FUNCTION_BLOCK FB_CYLINDER_DA_TESTDEV2_4 IMPLEMENTS I_CYLINDER_DA_TESTDEV2_4
VAR_INPUT
  bDoableActing:                                          BOOL;
  lrCurrentPosAbs:                                        LREAL;
  rCurrentPressureInBar:                                  REAL;
  rCurrentPressureInBarA:                                 REAL;
  rCurrentPressureInBarB:                                 REAL;
  /// Cylinder piston surface A
  lrPistonSurfaceA:                                       LREAL;
  /// Cylinder piston surface B
  lrPistonSurfaceB:                                       LREAL;
  // Speed and Pressure regulation
  rSpeedRegulationFactor:                                 REAL;
  rSpeedRegulationTolerance:                              REAL;
  rPressureRegulationFactor:                              REAL;
  rPressureRegulationTolerance:                           REAL;
END_VAR
VAR //General
	{attribute 'instance-path'} 
  {attribute 'noinit'} 
	strInstancePath:									                      STRING;
	bInit: 												                          BOOL:=TRUE;
	strFullObjectPath: 								                      STRING;
	stEvent:											                          ST_EVENT;
	bAck:												                            BOOL;
END_VAR
VAR   // From FB_init	
	itfLogEvents: 										                      I_HANDLE_EVENTS;
  itfOpMode:											                        I_OP_MODE;
  itfOpModeVisu:											                    I_OP_MODE_PAUSE_VISU;
  itfValve_CylCtrl:                                       I_VALVE_X_3_PROP;
  itfValve_LockA:                                         I_VALVE_X_2;
  itfValve_LockB:                                         I_VALVE_X_2;
  itfValve_PressureLimit:                                 I_PRV_PROP;
  rEndPosTol:                                             REAL;
  /// Volume flow in l/min or dm³/min
  rPumpVolumeFlow:                                        REAL; // Volumenstrom
  /// Pump efficiency factor (0,5-1)
  rPumpEfficiencyFactor:                                  REAL; // Wirkungsgrad
END_VAR                                      				
VAR	// Step chain control                				
  eSeq, eLastSeq, eNextSeq:					                      E_SEQ_CYLINDER; 
                  				
  //eActiveSeqState, eLastActiveSeqState:                 E_SEQ_GENERAL;
	(*
  iInternalSeqStateCase, iLastInternalSeqStateCase:       INT:=0;       
	tonDelay, tonTimeOut, tonStepTime:						          TON;
	tDelay:													                        TIME := T#100MS;
	tTimeOut:												                        TIME := T#100MS;
	tTimeOutExt:											                      TIME := T#100MS;
	bDelayActive, bTimeOutActiveQuit, bTimeOutActiveNoQuit:	BOOL;//Timer Option
	bActiveStep, bDebugAcitve, bDebugNext:					        BOOL;//Debug Option
	i:														                          INT;
 	iError:													                        INT; //ERROR-CODE                    	                   		
	listLastSteps:											                    ARRAY[0..49] OF ST_LAST_STEPS;	
	strExtraInfo:											                      STRING; 
	eStep_Type:												                      E_STEP_STATE_TYPE; 
	bDebugModeActive:										                    BOOL;   
	bWaitForBreakpoint:										                  BOOL;
	bBreakpointActive:										                  BOOL;
	bDebugResume:											                      BOOL;   
	listBreakpoint:											                    ARRAY[0..10] OF  INT;    
*)
i:														                            INT;
ii:														                            INT;
iii:														                          INT;
stSeqCtrlGeneral:											                    ST_SEQ_CTRL_GEN;     	
END_VAR                                             		
VAR                                                 		
	bMethodeFromExtStarted:									                BOOL;
	bMethodeFromExtActive:									                BOOL;
	bMethodeFromExtDone:									                  BOOL;
	strTemp:												                        STRING;
END_VAR   
VAR
  stHMI:                                                  ST_HMI_CYLINDER;
  lrToSetPos:                                             LREAL;
  rTargetPressureInBarA:                                  REAL;
  rTargetPressureInBarB:                                  REAL;
  rTargetPressureInForceA:                                REAL;
  rTargetPressureInForceB:                                REAL;
  rTargetPressureInPercentA:                              REAL;
  rTargetPressureInPercentB:                              REAL;
  iTargetPressureAsValueA:                                INT;
  iTargetPressureAsValueB:                                INT;
  rSpeedInPercentToSet:                                   REAL;
  rSpeedInMmPerSToSet:                                    REAL;
  rCurrentSpeedInMmPerS:                                  REAL;
  bStrokeLengthInitialized:                               BOOL;
  rStrokeLength:                                          REAL;
  lrPos:                                                  LREAL;
  lrPosZero:                                              LREAL;
  lrPosMax:                                               LREAL;
  bOpenChA:                                               BOOL;
	bOpenChB:                                               BOOL;
END_VAR
VAR // Recording
  stRecord:											                          ST_RECORD;	 
	tonSaveInterval:											                  TON; 
	iCntRecord:											                        INT;	
	listGainRampData:									                      ARRAY[0..499] OF stMesswerte;
	stCurrentRamp:										                      stRampAnalytic;
	iCycleCntNormal:									                      INT;	
	uiLinRegStart:										                      UINT:=0;
  uiLinRegEnd:										                        UINT:=299; 
  rGainLimit_EndPos:                                      REAL:=0.1;
  lrLastPos:                                              LREAL;
  bJogCtrlBusy:                                           BOOL;
  bStartHPTrigger:                                        BOOL;
  bStartWPTrigger:                                        BOOL;
  bStopTrigger:                                           BOOL;
  bStartCalibrationClicked:                               BOOL;
  // Speed
  listPosTable:                                           ARRAY[1..100] OF REAL;
  lrTotalPath:                                            LREAL;
  x:                                                      INT;
  xx:                                                     INT;
  iCorrectedSpeedValue:                                   INT;
  rCorrectedSpeedPercent:                                 REAL;
  bRegulation:                                            BOOL;
  bRegulationTrigger:                                     BOOL;
  uiRegulationSeq:                                        UINT := 0;
  bCorrectionTrigger:                                     BOOL;
  bRegulationBusy:                                        BOOL;
  rCurrentForceInKN:                                      REAL;
  rCurrentForceInN:                                       REAL;
  rActiveForce:                                           REAL;
  iCorrectedPressureAsValue:                              INT;
  bPressureRegulationTrigger:                             BOOL;
  bPressureRegulationBusy:                                BOOL;
  bPressureCorrectionTrigger:                             BOOL;
  uiPressureRegulationSeq:                                UINT := 0;
  bPressureRegulation:                                    BOOL;
END_VAR                	
VAR_TEMP                    	
	iTemp:										                              INT;
END_VAR
VAR PERSISTENT
	listCylCalibration:                                     ARRAY[1..2, 1..100] OF LREAL;
  listCalibrationTable:                                   ARRAY[1..7] OF ST_CYL_CALIBRATION;
END_VAR

// Set FBs and Interfaces ready after switch internal step
IF stSeqCtrlGeneral.iInternalSeqStateCase <> stSeqCtrlGeneral.iLastInternalSeqStateCase AND NOT stSeqCtrlGeneral.bExitSetReadyState THEN
  IF TRUE
  AND itfValve_CylCtrl.M_SetReady()
  AND itfValve_LockA.M_SetReady()
  AND itfValve_LockB.M_SetReady()
  AND itfValve_PressureLimit.M_SetReady()
  THEN
    stSeqCtrlGeneral.bExitSetReadyState := TRUE;
  ELSE
    RETURN;
  END_IF
END_IF

stSeqCtrlGeneral.strObjectPath := strInstancePath;
stSeqCtrlGeneral.strObject := F_CreateObjectName(strInstancePath);

rCurrentForceInKN := P_CurrentForceInKN;
rCurrentForceInN := P_CurrentForceInKN * 1000;

// First method call
_m_SequenceManager();
//_m_SaveLastStep();
_m_Recording();
_m_SpeedRegulation();
_m_PressureRegulation();
_m_PressureCalibration();
_m_HMI();

CASE eSeq OF 
  E_SEQ_CYLINDER.BASE:;
  
	E_SEQ_CYLINDER.INIT: _m_Seq_INIT();
		IF TRUE
		AND (stSeqCtrlGeneral.eActiveSeqState = E_SEQ_GENERAL.DONE) 
		THEN
			eSeq := E_SEQ_CYLINDER.BASE;
		END_IF
		
	E_SEQ_CYLINDER.SETUP:;
  
	// Process
  E_SEQ_CYLINDER.SET_MAX_POS: _m_Seq_SET_MAX_POS();
    IF TRUE
		AND (stSeqCtrlGeneral.eActiveSeqState = E_SEQ_GENERAL.DONE) 
		THEN
			eSeq := E_SEQ_CYLINDER.BASE;
		END_IF
  
  E_SEQ_CYLINDER.SET_WORK_PRESSURE: _m_Seq_SET_WORK_PRESSURE();
    IF TRUE
		AND (stSeqCtrlGeneral.eActiveSeqState = E_SEQ_GENERAL.DONE) 
		THEN
			eSeq := E_SEQ_CYLINDER.BASE;
		END_IF
  
  E_SEQ_CYLINDER.SET_ZERO_POS: _m_Seq_SET_ZERO_POS();
    IF TRUE
		AND (stSeqCtrlGeneral.eActiveSeqState = E_SEQ_GENERAL.DONE) 
		THEN
			eSeq := E_SEQ_CYLINDER.BASE;
		END_IF
  
  E_SEQ_CYLINDER.STOP: _m_Seq_STOP();
    IF TRUE
		AND (stSeqCtrlGeneral.eActiveSeqState = E_SEQ_GENERAL.DONE) 
		THEN
			eSeq := E_SEQ_CYLINDER.BASE;
		END_IF
    
  E_SEQ_CYLINDER.STOP_AND_LOCK: _m_Seq_STOP_AND_LOCK();
    IF TRUE
		AND (stSeqCtrlGeneral.eActiveSeqState = E_SEQ_GENERAL.DONE) 
		THEN
			eSeq := E_SEQ_CYLINDER.BASE;
		END_IF
  
  E_SEQ_CYLINDER.TO_HP: _m_Seq_TO_HP();
    IF TRUE
		AND (stSeqCtrlGeneral.eActiveSeqState = E_SEQ_GENERAL.DONE) 
		THEN
			eSeq := E_SEQ_CYLINDER.BASE;
		END_IF
  
  E_SEQ_CYLINDER.TO_SET_POS: _m_Seq_TO_SET_POS();
    IF TRUE
		AND (stSeqCtrlGeneral.eActiveSeqState = E_SEQ_GENERAL.DONE) 
		THEN
			eSeq := E_SEQ_CYLINDER.BASE;
		END_IF
  
  E_SEQ_CYLINDER.TO_WP: _m_Seq_TO_WP();
    IF TRUE
		AND (stSeqCtrlGeneral.eActiveSeqState = E_SEQ_GENERAL.DONE) 
		THEN
			eSeq := E_SEQ_CYLINDER.BASE;
		END_IF
    
  E_SEQ_CYLINDER.PRESSURE_CALIBRATION: _m_Seq_PRESSURE_CALIBRATION();
    IF TRUE
		AND (stSeqCtrlGeneral.eActiveSeqState = E_SEQ_GENERAL.DONE) 
		THEN
			eSeq := E_SEQ_CYLINDER.BASE;
		END_IF
    
  E_SEQ_CYLINDER.OPEN_LOCK_VALVES: _m_Seq_OPEN_LOCK_VALVES();
    IF TRUE
		AND (stSeqCtrlGeneral.eActiveSeqState = E_SEQ_GENERAL.DONE) 
		THEN
			eSeq := E_SEQ_CYLINDER.BASE;
		END_IF

  // End
	E_SEQ_CYLINDER.END:;
	E_SEQ_CYLINDER.ERROR_SEQ:;	
END_CASE

strTemp:=TO_STRING(eSeq);

METHOD PRIVATE _m_DebugManager
VAR_INPUT
	iStepID: int;
END_VAR
IF TRUE
AND THIS^.stSeqCtrlGeneral.bDebugModeActive 
AND NOT THIS^.stSeqCtrlGeneral.bActiveStep
THEN


THIS^.stSeqCtrlGeneral.bBreakpointActive:=FALSE;

FOR i:=0 TO 10 DO
	
	IF TRUE
	AND iStepID=THIS^.stSeqCtrlGeneral.listBreakpoint[i] 
	AND iStepID<>0
	THEN
		EXIT;
	END_IF
END_FOR
IF (i<=10) THEN
	THIS^.stSeqCtrlGeneral.bBreakpointActive:=TRUE;
END_IF

END_IF
END_METHOD

METHOD PRIVATE _m_Delay : BOOL
VAR_INPUT
	DelayTime:	TIME;
END_VAR
THIS^.stSeqCtrlGeneral.bDelayActive:=TRUE;
THIS^.stSeqCtrlGeneral.tDelay:=DelayTime;
_m_Delay:=FALSE;
IF THIS^.stSeqCtrlGeneral.tonDelay.Q THEN
	_m_Delay:=TRUE;
END_IF
END_METHOD

METHOD PRIVATE _m_GeneralStepSetting : BOOL
VAR_INPUT
	StepType:			    	E_STEP_STATE_TYPE;
	InfoTextID:					STRING(20);
	EnableDebug:	   			BOOL;	
	
END_VAR
IF THIS^.stSeqCtrlGeneral.bActiveStep THEN
	THIS^.stSeqCtrlGeneral.eStep_Type:=StepType;
	THIS^.stSeqCtrlGeneral.strExtraInfo:= GenLib.F_RET_TXTLIST_ENTRY(strPortNr:='851',strID:='',strTxtLstName:=InfoTextID);
END_IF
END_METHOD

METHOD PRIVATE _m_HMI : BOOL
VAR_INPUT
END_VAR
THIS^.stHMI.bInHP := THIS^.lrPos <= 1;
THIS^.stHMI.bInWP := THIS^.lrPos >= rStrokeLength - 1;
THIS^.stHMI.bPressureOk := THIS^.rCurrentPressureInBar > 25;
THIS^.stHMI.lrCurrentPos := THIS^.lrPos;
THIS^.stHMI.lrMaxPosVal := THIS^.lrPosMax;
THIS^.stHMI.lrMinPosVal := THIS^.lrPosZero;
THIS^.stHMI.sState := TO_STRING(THIS^.eSeq);
END_METHOD

METHOD PRIVATE _m_ManualOperation : BOOL
VAR_INPUT
END_VAR
IF TRUE 
AND THIS^.itfOpMode.P_OP_MODE_STATE = OP_MODE.MANUAL 
AND THIS^.itfOpModeVisu.P_HandSelected
AND THIS^.stHMI.bToHPTriggered
AND NOT THIS^.bJogCtrlBusy
THEN
  THIS^.stSeqCtrlGeneral.eActiveSeqState := E_SEQ_GENERAL.READY;
  THIS^.bStartHPTrigger := TRUE;
  THIS^.bJogCtrlBusy := TRUE;
ELSIF TRUE 
AND THIS^.itfOpMode.P_OP_MODE_STATE = OP_MODE.MANUAL 
AND THIS^.itfOpModeVisu.P_HandSelected
AND THIS^.stHMI.bToWPTriggered
AND NOT THIS^.bJogCtrlBusy
THEN
  THIS^.stSeqCtrlGeneral.eActiveSeqState := E_SEQ_GENERAL.READY;
  THIS^.bStartWPTrigger := TRUE;
  THIS^.bJogCtrlBusy := TRUE; 
ELSIF TRUE 
AND THIS^.itfOpMode.P_OP_MODE_STATE = OP_MODE.MANUAL 
AND THIS^.itfOpModeVisu.P_HandSelected
AND THIS^.stHMI.bToSetPosTriggered
AND NOT THIS^.bJogCtrlBusy
THEN
  //M_ToSetPos(lrToSetPos:= 500, rSpeedInPercent:= 100);
  THIS^.bJogCtrlBusy := TRUE;
ELSIF TRUE 
AND THIS^.itfOpMode.P_OP_MODE_STATE = OP_MODE.MANUAL 
AND THIS^.itfOpModeVisu.P_HandSelected
AND NOT THIS^.stHMI.bToHPTriggered
AND NOT THIS^.stHMI.bToWPTriggered
AND NOT THIS^.stHMI.bToSetPosTriggered
AND THIS^.bJogCtrlBusy
THEN
  THIS^.stSeqCtrlGeneral.eActiveSeqState := E_SEQ_GENERAL.READY;
  THIS^.bStopTrigger := TRUE;
  THIS^.bStartHPTrigger := FALSE;
  THIS^.bStartWPTrigger := FALSE;
  THIS^.bJogCtrlBusy := FALSE;
END_IF



IF THIS^.bStartWPTrigger THEN
  IF M_ToWP(ePressureType:= E_PRESSURE_TYPE.PERCENT, rWorkPressure:= 50, eSpeedType:= E_SPEED_TYPE.PERCENT, rSpeed:= 100) THEN
    THIS^.bStartWPTrigger := FALSE;
	END_IF
END_IF
IF THIS^.bStartHPTrigger THEN
  IF M_ToHP(ePressureType:= E_PRESSURE_TYPE.PERCENT, rWorkPressure:= 50, eSpeedType:= E_SPEED_TYPE.PERCENT, rSpeed:= 100) THEN
    THIS^.bStartHPTrigger := FALSE;
	END_IF
END_IF
IF THIS^.bStopTrigger THEN
  IF M_Stop() THEN
    THIS^.bStopTrigger := FALSE;
	END_IF
END_IF
END_METHOD

METHOD PRIVATE _m_PressureCalibration : BOOL
VAR_INPUT
END_VAR
// Calibration clicked
IF TRUE
AND THIS^.itfOpMode.P_OP_MODE_STATE = OP_MODE.MANUAL 
AND THIS^.bStartCalibrationClicked 
THEN
  IF M_PressureCalibration() THEN
    THIS^.stSeqCtrlGeneral.eActiveSeqState := E_SEQ_GENERAL.READY;
    THIS^.bStartCalibrationClicked := FALSE;
	END_IF
END_IF
END_METHOD

(******************Description****************)
// This function allows variable pressure control
(*********************************************)
METHOD PRIVATE _m_PressureRegulation : BOOL
VAR_INPUT
END_VAR
IF TRUE
AND THIS^.rCurrentForceInN < THIS^.rActiveForce 
AND THIS^.iCorrectedPressureAsValue < 32768
AND THIS^.bPressureRegulationTrigger
AND NOT THIS^.bPressureRegulationBusy
THEN
  IF ABS(THIS^.rCurrentForceInN - THIS^.rActiveForce) > THIS^.rPressureRegulationTolerance THEN
    //THIS^.iCorrectedPressureAsValue := THIS^.iCorrectedPressureAsValue + 100;
    THIS^.iCorrectedPressureAsValue := TO_INT(THIS^.iCorrectedPressureAsValue + ABS((THIS^.rCurrentForceInN - THIS^.rActiveForce) * THIS^.rPressureRegulationFactor));
    THIS^.bPressureCorrectionTrigger := TRUE;
  END_IF
ELSIF TRUE
AND THIS^.rCurrentForceInN > THIS^.rActiveForce 
AND THIS^.iCorrectedPressureAsValue > 0
AND THIS^.bPressureRegulationTrigger
AND NOT THIS^.bPressureRegulationBusy
THEN
  IF ABS(THIS^.rCurrentForceInN - THIS^.rActiveForce) > THIS^.rPressureRegulationTolerance THEN
    //THIS^.iCorrectedPressureAsValue := THIS^.iCorrectedPressureAsValue - 100;
    THIS^.iCorrectedPressureAsValue := TO_INT(THIS^.iCorrectedPressureAsValue - ABS((THIS^.rCurrentForceInN - THIS^.rActiveForce) * THIS^.rPressureRegulationFactor));
    THIS^.bPressureCorrectionTrigger := TRUE;
  END_IF
END_IF

// Set Valve value correction
IF THIS^.bPressureCorrectionTrigger THEN
  THIS^.bPressureRegulationBusy:= TRUE;
  CASE THIS^.uiPressureRegulationSeq OF
    0:;
      IF THIS^.itfValve_PressureLimit.M_SetReady() THEN
        THIS^.uiPressureRegulationSeq := 1;
	    END_IF
    1:;
      IF THIS^.itfValve_PressureLimit.M_SetLimit(ePressureType:= E_PRESSURE_TYPE.VALUE, rLimit:= iCorrectedPressureAsValue) THEN
        THIS^.bPressureCorrectionTrigger := FALSE;
        THIS^.bPressureRegulationBusy := FALSE;
        THIS^.uiPressureRegulationSeq := 0;
	    END_IF
	END_CASE
END_IF
END_METHOD

METHOD PRIVATE _m_Recording : BOOL
VAR_INPUT
END_VAR
VAR
	i:                      DINT;
END_VAR
// Recording data for 5s
tonSaveInterval(IN:= NOT tonSaveInterval.Q, pt:= T#100MS);

IF iCntRecord > 499 OR iCntRecord < 0 THEN
	iCntRecord := 0;
END_IF

IF THIS^.tonSaveInterval.Q THEN
	FOR i := 299 TO 1 BY -1 DO
		THIS^.stRecord.listRecordData[i].rPosition := THIS^.stRecord.listRecordData[i - 1].rPosition;	                                  		
		THIS^.stRecord.listRecordData[i].rPressureInBar := THIS^.stRecord.listRecordData[i - 1].rPressureInBar;
	END_FOR		

	// Messergebnisse in Array eintragen	
	THIS^.stRecord.listRecordData[i].rPosition :=	THIS^.lrPos;
	THIS^.stRecord.listRecordData[i].rPressureInBar := THIS^.rCurrentPressureInBar;
END_IF

// Calibration table
FOR THIS^.iii := 1 TO 7 BY 1 DO
  THIS^.listCylCalibration[2, THIS^.iii] := TO_LREAL(THIS^.listCalibrationTable[THIS^.iii].uiValue);
  THIS^.listCylCalibration[1, THIS^.iii] := TO_LREAL(THIS^.listCalibrationTable[THIS^.iii].uiPressure);
END_FOR

// Position
THIS^.lrPos := -(THIS^.lrCurrentPosAbs / 1000 - THIS^.lrPosZero);
THIS^.rStrokeLength := -(THIS^.lrPosMax - THIS^.lrPosZero);

// Speed
IF THIS^.x < 1 OR THIS^.x > 100 THEN
  THIS^.x := 1;
END_IF
THIS^.listPosTable[THIS^.x] := THIS^.lrPos - THIS^.lrLastPos;
THIS^.lrTotalPath := 0;
FOR THIS^.xx := 1 TO 100 BY 1 DO
  THIS^.lrTotalPath := THIS^.lrTotalPath + THIS^.listPosTable[THIS^.xx];
END_FOR
THIS^.rCurrentSpeedInMmPerS := THIS^.lrTotalPath;
THIS^.x := THIS^.x + 1;
THIS^.lrLastPos := THIS^.lrPos;
END_METHOD

METHOD PRIVATE _m_SaveLastStep : BOOL
VAR_INPUT
END_VAR
VAR
	i: dint;
END_VAR
IF NOT THIS^.stSeqCtrlGeneral.bActiveStep THEN
	
	FOR i:=49 TO 1 BY -1 DO
			stSeqCtrlGeneral.listLastSteps[i].strStepName:=stSeqCtrlGeneral.listLastSteps[i-1].strStepName;
			stSeqCtrlGeneral.listLastSteps[i].tStepTime:=stSeqCtrlGeneral.listLastSteps[i-1].tStepTime;
			stSeqCtrlGeneral.listLastSteps[i].tDelayTime:=stSeqCtrlGeneral.listLastSteps[i-1].tDelayTime;
	END_FOR
	stSeqCtrlGeneral.listLastSteps[0].strStepName:=TO_STRING(THIS^.eSeq);
	stSeqCtrlGeneral.listLastSteps[1].tStepTime:=THIS^.stSeqCtrlGeneral.tonStepTime.ET;
	stSeqCtrlGeneral.listLastSteps[1].tStepTime:=THIS^.stSeqCtrlGeneral.tonDelay.ET;
ELSE
	stSeqCtrlGeneral.listLastSteps[0].tStepTime:=THIS^.stSeqCtrlGeneral.tonStepTime.ET;
	stSeqCtrlGeneral.listLastSteps[0].tDelayTime:=THIS^.stSeqCtrlGeneral.tonDelay.ET;	
END_IF
END_METHOD

METHOD PRIVATE _m_Seq_INIT : E_SEQ_PROCESS
VAR_INPUT
END_VAR
VAR
	ActiveSeq: STRING;
END_VAR
VAR
	i:         INT;
END_VAR
//THIS^._m_GeneralStepSetting(StepType:=E_STEP_STATE_TYPE.INIT,
ActiveSeq := TO_STRING(THIS^.eSeq);

CASE THIS^.stSeqCtrlGeneral.eActiveSeqState OF
E_SEQ_GENERAL.READY:;

	
E_SEQ_GENERAL.EXECUTE:;
	IF TRUE
	THEN
		THIS^.stSeqCtrlGeneral.eActiveSeqState := E_SEQ_GENERAL.RESET;
	END_IF
E_SEQ_GENERAL.RESET:;
	stSeqCtrlGeneral.iInternalSeqStateCase := 0;
	IF TRUE
	THEN
		THIS^.stSeqCtrlGeneral.eActiveSeqState := E_SEQ_GENERAL.BUSY;
	END_IF
  
E_SEQ_GENERAL.BUSY:;
	CASE THIS^.stSeqCtrlGeneral.iInternalSeqStateCase OF
		0:	// Reset valves
      IF TRUE
      AND THIS^.itfValve_CylCtrl.M_Reset()
      AND THIS^.itfValve_LockA.M_ToHP(tDelay:= T#10MS)
      AND THIS^.itfValve_LockB.M_ToHP(tDelay:= T#10MS)
			THEN 
				THIS^.stSeqCtrlGeneral.iInternalSeqStateCase := 1000;
			END_IF
      
    1000: // Exit step
      IF TRUE
			THEN 
				THIS^.stSeqCtrlGeneral.iInternalSeqStateCase := 9999;
			END_IF
      
	ELSE
		THIS^.stSeqCtrlGeneral.eActiveSeqState := E_SEQ_GENERAL.DONE;  
	END_CASE
	THIS^.stSeqCtrlGeneral.strExtraInfo := CONCAT('Internal state: ', TO_STRING(THIS^.stSeqCtrlGeneral.iInternalSeqStateCase));
E_SEQ_GENERAL.DONE:;
E_SEQ_GENERAL.ERROR:;
E_SEQ_GENERAL.TIME_OUT:; 

IF TRUE
AND THIS^.stSeqCtrlGeneral.bTimeOutActiveQuit 
THEN
  THIS^.stSeqCtrlGeneral.strExtraInfo := 'Bitte quittieren und erneut testen';
  IF TRUE
  //AND itfOpMode.P_QUIT
  THEN
    THIS^.stSeqCtrlGeneral.eActiveSeqState := E_SEQ_GENERAL.EXECUTE;
	END_IF
  
END_IF

ELSE
  THIS^.stSeqCtrlGeneral.eActiveSeqState := E_SEQ_GENERAL.ERROR;
END_CASE
END_METHOD

METHOD PRIVATE _m_Seq_OPEN_LOCK_VALVES : E_SEQ_PROCESS
VAR_INPUT
END_VAR
VAR
	ActiveSeq: STRING;
END_VAR
VAR
	
END_VAR
//THIS^._m_GeneralStepSetting(StepType:=E_STEP_STATE_TYPE.INIT,
ActiveSeq := TO_STRING(THIS^.eSeq);

CASE THIS^.stSeqCtrlGeneral.eActiveSeqState OF
E_SEQ_GENERAL.READY:;

	
E_SEQ_GENERAL.EXECUTE:;
	IF TRUE
	THEN
		THIS^.stSeqCtrlGeneral.eActiveSeqState := E_SEQ_GENERAL.RESET;
	END_IF
  
E_SEQ_GENERAL.RESET:;
	stSeqCtrlGeneral.iInternalSeqStateCase := 0;
	IF TRUE
	THEN
		THIS^.stSeqCtrlGeneral.eActiveSeqState := E_SEQ_GENERAL.BUSY;
	END_IF
  
E_SEQ_GENERAL.BUSY:;
	CASE THIS^.stSeqCtrlGeneral.iInternalSeqStateCase OF
    0:	// Check if open A
      IF TRUE
			THEN 
        IF THIS^.bOpenChA THEN
          THIS^.stSeqCtrlGeneral.iInternalSeqStateCase := 10;
        ELSE
          THIS^.stSeqCtrlGeneral.iInternalSeqStateCase := 20;
        END_IF
			END_IF

    10:	// Open A
      IF TRUE 
      AND THIS^.itfValve_LockA.M_ToWP1(tDelay:= T#0MS)
			THEN 
        THIS^.stSeqCtrlGeneral.iInternalSeqStateCase := 30;
			END_IF
      
		20:	// Close A
      IF TRUE
      AND THIS^.itfValve_LockA.M_ToHP(tDelay:= T#0MS)
			THEN 
        THIS^.stSeqCtrlGeneral.iInternalSeqStateCase := 30;
			END_IF
      
    30:	// Check if open B
      IF TRUE
			THEN 
        IF THIS^.bOpenChB THEN
          THIS^.stSeqCtrlGeneral.iInternalSeqStateCase := 40;
        ELSE
          THIS^.stSeqCtrlGeneral.iInternalSeqStateCase := 50;
        END_IF
			END_IF

    40:	// Open B
      IF TRUE
      AND THIS^.itfValve_LockB.M_ToWP1(tDelay:= T#0MS)
			THEN 
        THIS^.stSeqCtrlGeneral.iInternalSeqStateCase := 1000;
			END_IF
      
		50:	// Close B
      IF TRUE
      AND THIS^.itfValve_LockB.M_ToHP(tDelay:= T#0MS)
			THEN 
        THIS^.stSeqCtrlGeneral.iInternalSeqStateCase := 1000;
			END_IF
      
    1000: // Exit step
      IF TRUE
			THEN 
				THIS^.stSeqCtrlGeneral.iInternalSeqStateCase := 9999;
			END_IF
      
	ELSE
		THIS^.stSeqCtrlGeneral.eActiveSeqState := E_SEQ_GENERAL.DONE;  
	END_CASE
	THIS^.stSeqCtrlGeneral.strExtraInfo := CONCAT('Internal state: ', TO_STRING(THIS^.stSeqCtrlGeneral.iInternalSeqStateCase));

E_SEQ_GENERAL.DONE:;

E_SEQ_GENERAL.ERROR:;

E_SEQ_GENERAL.TIME_OUT:; 
IF TRUE
AND THIS^.stSeqCtrlGeneral.bTimeOutActiveQuit 
THEN
  THIS^.stSeqCtrlGeneral.strExtraInfo := 'Bitte quittieren und erneut testen';
  IF TRUE
  //AND itfOpMode.P_QUIT
  THEN
    THIS^.stSeqCtrlGeneral.eActiveSeqState := E_SEQ_GENERAL.EXECUTE;
	END_IF
  
END_IF

ELSE
  THIS^.stSeqCtrlGeneral.eActiveSeqState := E_SEQ_GENERAL.ERROR;
END_CASE
END_METHOD

METHOD PRIVATE _m_Seq_PRESSURE_CALIBRATION : E_SEQ_PROCESS
VAR_INPUT
END_VAR
VAR
	ActiveSeq:  STRING;
END_VAR
//THIS^._m_GeneralStepSetting(StepType:=E_STEP_STATE_TYPE.INIT,
ActiveSeq := TO_STRING(THIS^.eSeq);

CASE THIS^.stSeqCtrlGeneral.eActiveSeqState OF
E_SEQ_GENERAL.READY:;

	
E_SEQ_GENERAL.EXECUTE:;
	IF TRUE
	THEN
		THIS^.stSeqCtrlGeneral.eActiveSeqState := E_SEQ_GENERAL.RESET;
	END_IF
  
E_SEQ_GENERAL.RESET:;
	stSeqCtrlGeneral.iInternalSeqStateCase := 0;
	IF TRUE
	THEN
    THIS^.ii := 1;
    FOR THIS^.ii := 1 TO 7 BY 1 DO
      THIS^.listCalibrationTable[THIS^.ii].uiValue := 0;
      THIS^.listCalibrationTable[THIS^.ii].uiPressure := 0;
      THIS^.listCalibrationTable[THIS^.ii].uiState := 0;
		END_FOR
    THIS^.ii := 1;
		THIS^.stSeqCtrlGeneral.eActiveSeqState := E_SEQ_GENERAL.BUSY;
	END_IF
  
E_SEQ_GENERAL.BUSY:;
	CASE THIS^.stSeqCtrlGeneral.iInternalSeqStateCase OF
		0:	// Set work pressure value to XXXX
      IF TRUE
      AND THIS^.itfValve_PressureLimit.M_SetLimit(ePressureType:= E_PRESSURE_TYPE.VALUE, rLimit:= 1000 * THIS^.ii)
			THEN 
        THIS^.listCalibrationTable[THIS^.ii].uiValue := TO_UINT(1000 * THIS^.ii);
        THIS^.listCalibrationTable[THIS^.ii].uiState := 1;
        THIS^.stSeqCtrlGeneral.iInternalSeqStateCase := 10;
			END_IF
      
    10:	// Open A channel
      IF TRUE
      AND THIS^.itfValve_LockA.M_ToWP1(tDelay:= T#10MS)
			THEN 
        IF THIS^.bDoableActing THEN
				  THIS^.stSeqCtrlGeneral.iInternalSeqStateCase := 20;
        ELSE
          THIS^.stSeqCtrlGeneral.iInternalSeqStateCase := 30;
        END_IF
			END_IF
      
    20:	// Open B channel
      IF TRUE
      AND THIS^.itfValve_LockB.M_ToWP1(tDelay:= T#10MS)
			THEN 
				THIS^.stSeqCtrlGeneral.iInternalSeqStateCase := 30;
			END_IF
      
    30: // Move cylinder to WP
      IF TRUE
      AND THIS^.itfValve_CylCtrl.M_ValveCtrl(rSpeedInPercent:= 100, tDelay:= T#10MS)
			THEN 
        THIS^.stSeqCtrlGeneral.iInternalSeqStateCase := 40;
			END_IF
      
    40: // Choice step
      IF TRUE
      THEN
        IF THIS^.ii = 1 THEN
          THIS^.stSeqCtrlGeneral.iInternalSeqStateCase := 50;
        ELSE
          THIS^.stSeqCtrlGeneral.iInternalSeqStateCase := 60;
				END_IF
			END_IF
      
    50: // Delay step (wait for cylinder end position)
      IF TRUE
      AND _m_Delay(DelayTime:= T#30S)
      THEN
        THIS^.stSeqCtrlGeneral.iInternalSeqStateCase := 60;
			END_IF
      
    60: // Delay step (cylinder under load)
      IF TRUE
      AND _m_Delay(DelayTime:= T#5S)
      THEN
        THIS^.stSeqCtrlGeneral.iInternalSeqStateCase := 70;
			END_IF
      
    70: // Save pressure
      IF TRUE
      THEN
        THIS^.listCalibrationTable[THIS^.ii].uiPressure := TO_UINT(THIS^.rCurrentPressureInBar);
        THIS^.listCalibrationTable[THIS^.ii].uiState := 2;
        THIS^.stSeqCtrlGeneral.iInternalSeqStateCase := 80;
			END_IF
      
    80: // Decide step
      IF TRUE
      AND _m_Delay(DelayTime:= T#1S)
      THEN
        IF THIS^.ii >= 7 OR THIS^.ii < 1 THEN
          THIS^.ii := 1;
          THIS^.stSeqCtrlGeneral.iInternalSeqStateCase := 1000;
        ELSE
          THIS^.ii := THIS^.ii + 1;
          THIS^.stSeqCtrlGeneral.iInternalSeqStateCase := 0;
				END_IF
			END_IF
      
    1000: // Stop and exit
      IF TRUE
      AND THIS^.itfValve_PressureLimit.M_SetLimit(ePressureType:= E_PRESSURE_TYPE.VALUE, rLimit:= 0)
      AND THIS^.itfValve_CylCtrl.M_ValveCtrl(rSpeedInPercent:= 0, tDelay:= T#10MS)
      AND THIS^.itfValve_LockA.M_ToHP(tDelay:= T#10MS)
      AND THIS^.itfValve_LockB.M_ToHP(tDelay:= T#10MS)
			THEN 
				THIS^.stSeqCtrlGeneral.iInternalSeqStateCase := 9999;
			END_IF
      
	ELSE
		THIS^.stSeqCtrlGeneral.eActiveSeqState := E_SEQ_GENERAL.DONE;  
	END_CASE
	THIS^.stSeqCtrlGeneral.strExtraInfo := CONCAT('Internal state: ', TO_STRING(THIS^.stSeqCtrlGeneral.iInternalSeqStateCase));

E_SEQ_GENERAL.DONE:;

E_SEQ_GENERAL.ERROR:;

E_SEQ_GENERAL.TIME_OUT:; 
IF TRUE
AND THIS^.stSeqCtrlGeneral.bTimeOutActiveQuit 
THEN
  THIS^.stSeqCtrlGeneral.strExtraInfo := 'Bitte quittieren und erneut testen';
  IF TRUE
  //AND itfOpMode.P_QUIT
  THEN
    THIS^.stSeqCtrlGeneral.eActiveSeqState := E_SEQ_GENERAL.EXECUTE;
	END_IF
  
END_IF

ELSE
  THIS^.stSeqCtrlGeneral.eActiveSeqState := E_SEQ_GENERAL.ERROR;
END_CASE
END_METHOD

METHOD PRIVATE _m_Seq_SET_MAX_POS : E_SEQ_PROCESS
VAR_INPUT
END_VAR
VAR
	ActiveSeq: STRING;
END_VAR
VAR
	
END_VAR
//THIS^._m_GeneralStepSetting(StepType:=E_STEP_STATE_TYPE.INIT,
ActiveSeq := TO_STRING(THIS^.eSeq);

CASE THIS^.stSeqCtrlGeneral.eActiveSeqState OF
E_SEQ_GENERAL.READY:;

	
E_SEQ_GENERAL.EXECUTE:;
	IF TRUE
	THEN
		THIS^.stSeqCtrlGeneral.eActiveSeqState := E_SEQ_GENERAL.RESET;
	END_IF
  
E_SEQ_GENERAL.RESET:;
	stSeqCtrlGeneral.iInternalSeqStateCase := 0;
	IF TRUE
	THEN
		THIS^.stSeqCtrlGeneral.eActiveSeqState := E_SEQ_GENERAL.BUSY;
	END_IF
  
E_SEQ_GENERAL.BUSY:;
	CASE THIS^.stSeqCtrlGeneral.iInternalSeqStateCase OF
		0:	// Set max position
      IF TRUE 
			THEN 
        THIS^.lrPosMax := THIS^.lrCurrentPosAbs / 1000;
        THIS^.stSeqCtrlGeneral.iInternalSeqStateCase := 1000;
			END_IF
      
    1000: // Exit step
      IF TRUE
			THEN 
				THIS^.stSeqCtrlGeneral.iInternalSeqStateCase := 9999;
			END_IF
      
	ELSE
		THIS^.stSeqCtrlGeneral.eActiveSeqState := E_SEQ_GENERAL.DONE;  
	END_CASE
	THIS^.stSeqCtrlGeneral.strExtraInfo := CONCAT('Internal state: ', TO_STRING(THIS^.stSeqCtrlGeneral.iInternalSeqStateCase));

E_SEQ_GENERAL.DONE:;

E_SEQ_GENERAL.ERROR:;

E_SEQ_GENERAL.TIME_OUT:; 
IF TRUE
AND THIS^.stSeqCtrlGeneral.bTimeOutActiveQuit 
THEN
  THIS^.stSeqCtrlGeneral.strExtraInfo := 'Bitte quittieren und erneut testen';
  IF TRUE
  //AND itfOpMode.P_QUIT
  THEN
    THIS^.stSeqCtrlGeneral.eActiveSeqState := E_SEQ_GENERAL.EXECUTE;
	END_IF
  
END_IF

ELSE
  THIS^.stSeqCtrlGeneral.eActiveSeqState := E_SEQ_GENERAL.ERROR;
END_CASE
END_METHOD

METHOD PRIVATE _m_Seq_SET_WORK_PRESSURE : E_SEQ_PROCESS
VAR_INPUT
END_VAR
VAR
	ActiveSeq: STRING;
END_VAR
VAR
	
END_VAR
//THIS^._m_GeneralStepSetting(StepType:=E_STEP_STATE_TYPE.INIT,
ActiveSeq := TO_STRING(THIS^.eSeq);

CASE THIS^.stSeqCtrlGeneral.eActiveSeqState OF
E_SEQ_GENERAL.READY:;

	
E_SEQ_GENERAL.EXECUTE:;
	IF TRUE
	THEN
		THIS^.stSeqCtrlGeneral.eActiveSeqState := E_SEQ_GENERAL.RESET;
	END_IF
  
E_SEQ_GENERAL.RESET:;
	stSeqCtrlGeneral.iInternalSeqStateCase := 0;
	IF TRUE
	THEN
		THIS^.stSeqCtrlGeneral.eActiveSeqState := E_SEQ_GENERAL.BUSY;
	END_IF
  
E_SEQ_GENERAL.BUSY:;
	CASE THIS^.stSeqCtrlGeneral.iInternalSeqStateCase OF
		0:	// Set work pressure
      IF TRUE
      AND THIS^.itfValve_PressureLimit.M_SetLimit(ePressureType:= E_PRESSURE_TYPE.VALUE, rLimit:= TO_REAL(THIS^.iTargetPressureAsValueA))
			THEN 
        THIS^.stSeqCtrlGeneral.iInternalSeqStateCase := 1000;
			END_IF
      
    1000: // Exit step
      IF TRUE
			THEN 
				THIS^.stSeqCtrlGeneral.iInternalSeqStateCase := 9999;
			END_IF
      
	ELSE
		THIS^.stSeqCtrlGeneral.eActiveSeqState := E_SEQ_GENERAL.DONE;  
	END_CASE
	THIS^.stSeqCtrlGeneral.strExtraInfo := CONCAT('Internal state: ', TO_STRING(THIS^.stSeqCtrlGeneral.iInternalSeqStateCase));

E_SEQ_GENERAL.DONE:;

E_SEQ_GENERAL.ERROR:;

E_SEQ_GENERAL.TIME_OUT:; 
IF TRUE
AND THIS^.stSeqCtrlGeneral.bTimeOutActiveQuit 
THEN
  THIS^.stSeqCtrlGeneral.strExtraInfo := 'Bitte quittieren und erneut testen';
  IF TRUE
  //AND itfOpMode.P_QUIT
  THEN
    THIS^.stSeqCtrlGeneral.eActiveSeqState := E_SEQ_GENERAL.EXECUTE;
	END_IF
  
END_IF

ELSE
  THIS^.stSeqCtrlGeneral.eActiveSeqState := E_SEQ_GENERAL.ERROR;
END_CASE
END_METHOD

METHOD PRIVATE _m_Seq_SET_ZERO_POS : E_SEQ_PROCESS
VAR_INPUT
END_VAR
VAR
	ActiveSeq: STRING;
END_VAR
VAR
	
END_VAR
//THIS^._m_GeneralStepSetting(StepType:=E_STEP_STATE_TYPE.INIT,
ActiveSeq := TO_STRING(THIS^.eSeq);

CASE THIS^.stSeqCtrlGeneral.eActiveSeqState OF
E_SEQ_GENERAL.READY:;

	
E_SEQ_GENERAL.EXECUTE:;
	IF TRUE
	THEN
		THIS^.stSeqCtrlGeneral.eActiveSeqState := E_SEQ_GENERAL.RESET;
	END_IF
  
E_SEQ_GENERAL.RESET:;
	stSeqCtrlGeneral.iInternalSeqStateCase := 0;
	IF TRUE
	THEN
		THIS^.stSeqCtrlGeneral.eActiveSeqState := E_SEQ_GENERAL.BUSY;
	END_IF
  
E_SEQ_GENERAL.BUSY:;
	CASE THIS^.stSeqCtrlGeneral.iInternalSeqStateCase OF
		0:	// Set zero position
      IF TRUE 
			THEN 
        THIS^.lrPosZero := THIS^.lrCurrentPosAbs / 1000;
        THIS^.stSeqCtrlGeneral.iInternalSeqStateCase := 1000;
			END_IF
      
    1000: // Exit step
      IF TRUE
			THEN 
				THIS^.stSeqCtrlGeneral.iInternalSeqStateCase := 9999;
			END_IF
      
	ELSE
		THIS^.stSeqCtrlGeneral.eActiveSeqState := E_SEQ_GENERAL.DONE;  
	END_CASE
	THIS^.stSeqCtrlGeneral.strExtraInfo := CONCAT('Internal state: ', TO_STRING(THIS^.stSeqCtrlGeneral.iInternalSeqStateCase));

E_SEQ_GENERAL.DONE:;

E_SEQ_GENERAL.ERROR:;

E_SEQ_GENERAL.TIME_OUT:; 
IF TRUE
AND THIS^.stSeqCtrlGeneral.bTimeOutActiveQuit 
THEN
  THIS^.stSeqCtrlGeneral.strExtraInfo := 'Bitte quittieren und erneut testen';
  IF TRUE
  //AND itfOpMode.P_QUIT
  THEN
    THIS^.stSeqCtrlGeneral.eActiveSeqState := E_SEQ_GENERAL.EXECUTE;
	END_IF
  
END_IF

ELSE
  THIS^.stSeqCtrlGeneral.eActiveSeqState := E_SEQ_GENERAL.ERROR;
END_CASE
END_METHOD

METHOD PRIVATE _m_Seq_STOP : E_SEQ_PROCESS
VAR_INPUT
END_VAR
VAR
	ActiveSeq: STRING;
END_VAR
VAR
	
END_VAR
//THIS^._m_GeneralStepSetting(StepType:=E_STEP_STATE_TYPE.INIT,
ActiveSeq := TO_STRING(THIS^.eSeq);

CASE THIS^.stSeqCtrlGeneral.eActiveSeqState OF
E_SEQ_GENERAL.READY:;

	
E_SEQ_GENERAL.EXECUTE:;
	IF TRUE
	THEN
    THIS^.bRegulationTrigger := FALSE;
    THIS^.bPressureRegulationTrigger := FALSE;
		THIS^.stSeqCtrlGeneral.eActiveSeqState := E_SEQ_GENERAL.RESET;
	END_IF
  
E_SEQ_GENERAL.RESET:;
	stSeqCtrlGeneral.iInternalSeqStateCase := 0;
	IF TRUE
	THEN
		THIS^.stSeqCtrlGeneral.eActiveSeqState := E_SEQ_GENERAL.BUSY;
	END_IF
  
E_SEQ_GENERAL.BUSY:;
	CASE THIS^.stSeqCtrlGeneral.iInternalSeqStateCase OF
		0: // Switch off valves
      IF TRUE
      AND THIS^.itfValve_CylCtrl.M_ValveCtrl(rSpeedInPercent:= 0, tDelay:= T#0MS)
			THEN 
				THIS^.stSeqCtrlGeneral.iInternalSeqStateCase := 1000;
			END_IF
      
    1000: // Exit step
      IF TRUE
			THEN 
				THIS^.stSeqCtrlGeneral.iInternalSeqStateCase := 9999;
			END_IF
      
	ELSE
		THIS^.stSeqCtrlGeneral.eActiveSeqState := E_SEQ_GENERAL.DONE;  
	END_CASE
	THIS^.stSeqCtrlGeneral.strExtraInfo := CONCAT('Internal state: ', TO_STRING(THIS^.stSeqCtrlGeneral.iInternalSeqStateCase));

E_SEQ_GENERAL.DONE:;

E_SEQ_GENERAL.ERROR:;

E_SEQ_GENERAL.TIME_OUT:; 
IF TRUE
AND THIS^.stSeqCtrlGeneral.bTimeOutActiveQuit 
THEN
  THIS^.stSeqCtrlGeneral.strExtraInfo := 'Bitte quittieren und erneut testen';
  IF TRUE
  //AND itfOpMode.P_QUIT
  THEN
    THIS^.stSeqCtrlGeneral.eActiveSeqState := E_SEQ_GENERAL.EXECUTE;
	END_IF
  
END_IF

ELSE
  THIS^.stSeqCtrlGeneral.eActiveSeqState := E_SEQ_GENERAL.ERROR;
END_CASE
END_METHOD

METHOD PRIVATE _m_Seq_STOP_AND_LOCK : E_SEQ_PROCESS
VAR_INPUT
END_VAR
VAR
	ActiveSeq: STRING;
END_VAR
VAR
	
END_VAR
//THIS^._m_GeneralStepSetting(StepType:=E_STEP_STATE_TYPE.INIT,
ActiveSeq := TO_STRING(THIS^.eSeq);

CASE THIS^.stSeqCtrlGeneral.eActiveSeqState OF
E_SEQ_GENERAL.READY:;

	
E_SEQ_GENERAL.EXECUTE:;
	IF TRUE
	THEN
    THIS^.bRegulationTrigger := FALSE;
    THIS^.bPressureRegulationTrigger := FALSE;
		THIS^.stSeqCtrlGeneral.eActiveSeqState := E_SEQ_GENERAL.RESET;
	END_IF
  
E_SEQ_GENERAL.RESET:;
	stSeqCtrlGeneral.iInternalSeqStateCase := 0;
	IF TRUE
	THEN
		THIS^.stSeqCtrlGeneral.eActiveSeqState := E_SEQ_GENERAL.BUSY;
	END_IF
  
E_SEQ_GENERAL.BUSY:;
	CASE THIS^.stSeqCtrlGeneral.iInternalSeqStateCase OF
		0: // Switch off valves
      IF TRUE
      AND THIS^.itfValve_CylCtrl.M_ValveCtrl(rSpeedInPercent:= 0, tDelay:= T#0MS)
      AND THIS^.itfValve_LockA.M_ToHP(tDelay:= T#0MS)
      AND THIS^.itfValve_LockB.M_ToHP(tDelay:= T#0MS)
			THEN 
				THIS^.stSeqCtrlGeneral.iInternalSeqStateCase := 1000;
			END_IF
      
    1000: // Exit step
      IF TRUE
			THEN 
				THIS^.stSeqCtrlGeneral.iInternalSeqStateCase := 9999;
			END_IF
      
	ELSE
		THIS^.stSeqCtrlGeneral.eActiveSeqState := E_SEQ_GENERAL.DONE;  
	END_CASE
	THIS^.stSeqCtrlGeneral.strExtraInfo := CONCAT('Internal state: ', TO_STRING(THIS^.stSeqCtrlGeneral.iInternalSeqStateCase));

E_SEQ_GENERAL.DONE:;

E_SEQ_GENERAL.ERROR:;

E_SEQ_GENERAL.TIME_OUT:; 
IF TRUE
AND THIS^.stSeqCtrlGeneral.bTimeOutActiveQuit 
THEN
  THIS^.stSeqCtrlGeneral.strExtraInfo := 'Bitte quittieren und erneut testen';
  IF TRUE
  //AND itfOpMode.P_QUIT
  THEN
    THIS^.stSeqCtrlGeneral.eActiveSeqState := E_SEQ_GENERAL.EXECUTE;
	END_IF
  
END_IF

ELSE
  THIS^.stSeqCtrlGeneral.eActiveSeqState := E_SEQ_GENERAL.ERROR;
END_CASE
END_METHOD

METHOD PRIVATE _m_Seq_TO_HP : E_SEQ_PROCESS
VAR_INPUT
END_VAR
VAR
	ActiveSeq: STRING;
END_VAR
//THIS^._m_GeneralStepSetting(StepType:=E_STEP_STATE_TYPE.INIT,
ActiveSeq := TO_STRING(THIS^.eSeq);

CASE THIS^.stSeqCtrlGeneral.eActiveSeqState OF
E_SEQ_GENERAL.READY:;

	
E_SEQ_GENERAL.EXECUTE:;
	IF TRUE
	THEN
    THIS^.bRegulationTrigger := FALSE;
    THIS^.bPressureRegulationTrigger := FALSE;
		THIS^.stSeqCtrlGeneral.eActiveSeqState := E_SEQ_GENERAL.RESET;
	END_IF
  
E_SEQ_GENERAL.RESET:;
	stSeqCtrlGeneral.iInternalSeqStateCase := 0;
	IF TRUE
	THEN
		THIS^.stSeqCtrlGeneral.eActiveSeqState := E_SEQ_GENERAL.BUSY;
	END_IF
  
E_SEQ_GENERAL.BUSY:;
	CASE THIS^.stSeqCtrlGeneral.iInternalSeqStateCase OF
		0:	// Set work pressure
      IF TRUE
      AND THIS^.itfValve_PressureLimit.M_SetLimit(ePressureType:= E_PRESSURE_TYPE.VALUE, rLimit:= TO_REAL(THIS^.iTargetPressureAsValueB))
			THEN 
        THIS^.stSeqCtrlGeneral.iInternalSeqStateCase := 10;
			END_IF
    
    10:	// Switch on lock A valve
      IF TRUE
      AND THIS^.itfValve_LockA.M_ToWP1(tDelay:= T#0MS)
			THEN 
        IF THIS^.bDoableActing THEN
          THIS^.stSeqCtrlGeneral.iInternalSeqStateCase := 20;
        ELSE
          THIS^.stSeqCtrlGeneral.iInternalSeqStateCase := 30;
        END_IF
			END_IF
      
    20:	// Switch on lock B valve
      IF TRUE
      AND THIS^.itfValve_LockB.M_ToWP1(tDelay:= T#0MS)
			THEN 
        THIS^.stSeqCtrlGeneral.iInternalSeqStateCase := 30;
			END_IF
      
    30:	// Set valve control
      IF TRUE
      AND THIS^.itfValve_CylCtrl.M_ValveCtrl(rSpeedInPercent:= THIS^.rSpeedInPercentToSet, tDelay:= T#0MS)
			THEN 
        THIS^.stSeqCtrlGeneral.iInternalSeqStateCase := 1000;
			END_IF
      
    1000: // Exit step
      IF TRUE
			THEN 
				THIS^.stSeqCtrlGeneral.iInternalSeqStateCase := 9999;
			END_IF
      
	ELSE
		THIS^.stSeqCtrlGeneral.eActiveSeqState := E_SEQ_GENERAL.DONE;  
	END_CASE
	THIS^.stSeqCtrlGeneral.strExtraInfo := CONCAT('Internal state: ', TO_STRING(THIS^.stSeqCtrlGeneral.iInternalSeqStateCase));

E_SEQ_GENERAL.DONE:;
  THIS^.bRegulationTrigger := THIS^.bRegulation;
  THIS^.bPressureRegulationTrigger := THIS^.bPressureRegulation;

E_SEQ_GENERAL.ERROR:;

E_SEQ_GENERAL.TIME_OUT:; 
IF TRUE
AND THIS^.stSeqCtrlGeneral.bTimeOutActiveQuit 
THEN
  THIS^.stSeqCtrlGeneral.strExtraInfo := 'Bitte quittieren und erneut testen';
  IF TRUE
  //AND itfOpMode.P_QUIT
  THEN
    THIS^.stSeqCtrlGeneral.eActiveSeqState := E_SEQ_GENERAL.EXECUTE;
	END_IF
  
END_IF

ELSE
  THIS^.stSeqCtrlGeneral.eActiveSeqState := E_SEQ_GENERAL.ERROR;
END_CASE
END_METHOD

METHOD PRIVATE _m_Seq_TO_SET_POS : E_SEQ_PROCESS
VAR_INPUT
END_VAR
VAR
	ActiveSeq: STRING;
END_VAR
VAR
	
END_VAR
//THIS^._m_GeneralStepSetting(StepType:=E_STEP_STATE_TYPE.INIT,
ActiveSeq := TO_STRING(THIS^.eSeq);

CASE THIS^.stSeqCtrlGeneral.eActiveSeqState OF
E_SEQ_GENERAL.READY:;

	
E_SEQ_GENERAL.EXECUTE:;
	IF TRUE
	THEN
		THIS^.stSeqCtrlGeneral.eActiveSeqState := E_SEQ_GENERAL.RESET;
	END_IF
  
E_SEQ_GENERAL.RESET:;
	stSeqCtrlGeneral.iInternalSeqStateCase := 0;
	IF TRUE
	THEN
		THIS^.stSeqCtrlGeneral.eActiveSeqState := E_SEQ_GENERAL.BUSY;
	END_IF
  
E_SEQ_GENERAL.BUSY:;
	CASE THIS^.stSeqCtrlGeneral.iInternalSeqStateCase OF
		0:	// Switch valves
      IF TRUE
      AND THIS^.itfValve_LockA.M_ToWP1(tDelay:= T#10MS)
      AND THIS^.itfValve_LockB.M_ToWP1(tDelay:= T#10MS)
			THEN 
        IF bStrokeLengthInitialized 
        AND THIS^.lrToSetPos <= THIS^.rStrokeLength 
        AND THIS^.lrToSetPos >= 0.0 
        THEN
          // Set direction
          IF THIS^.lrPos > THIS^.lrToSetPos THEN
            THIS^.rSpeedInPercentToSet := -ABS(THIS^.rSpeedInPercentToSet);
			    END_IF
          THIS^.stSeqCtrlGeneral.iInternalSeqStateCase := 10;
        ELSE
          THIS^.stSeqCtrlGeneral.eActiveSeqState := E_SEQ_GENERAL.ERROR;
				END_IF
			END_IF
      
    10: // Move cylinder to HP and wait for endposition
      IF TRUE
      AND THIS^.itfValve_CylCtrl.M_ValveCtrl(rSpeedInPercent:= THIS^.rSpeedInPercentToSet, tDelay:= T#10MS)
			THEN 
        IF THIS^.lrPos < THIS^.rEndPosTol THEN
				  THIS^.stSeqCtrlGeneral.iInternalSeqStateCase := 20;
        END_IF
			END_IF
      
    20: // Switch off valves
      IF TRUE
      AND THIS^.itfValve_CylCtrl.M_ValveCtrl(rSpeedInPercent:= 0, tDelay:= T#10MS)
			THEN 
				THIS^.stSeqCtrlGeneral.iInternalSeqStateCase := 1000;
			END_IF
      
    1000: // Exit step
      IF TRUE
			THEN 
				THIS^.stSeqCtrlGeneral.iInternalSeqStateCase := 9999;
			END_IF
      
	ELSE
		THIS^.stSeqCtrlGeneral.eActiveSeqState := E_SEQ_GENERAL.DONE;  
	END_CASE
	THIS^.stSeqCtrlGeneral.strExtraInfo := CONCAT('Internal state: ', TO_STRING(THIS^.stSeqCtrlGeneral.iInternalSeqStateCase));

E_SEQ_GENERAL.DONE:;

E_SEQ_GENERAL.ERROR:;

E_SEQ_GENERAL.TIME_OUT:; 
IF TRUE
AND THIS^.stSeqCtrlGeneral.bTimeOutActiveQuit 
THEN
  THIS^.stSeqCtrlGeneral.strExtraInfo := 'Bitte quittieren und erneut testen';
  IF TRUE
  //AND itfOpMode.P_QUIT
  THEN
    THIS^.stSeqCtrlGeneral.eActiveSeqState := E_SEQ_GENERAL.EXECUTE;
	END_IF
  
END_IF

ELSE
  THIS^.stSeqCtrlGeneral.eActiveSeqState := E_SEQ_GENERAL.ERROR;
END_CASE
END_METHOD

METHOD PRIVATE _m_Seq_TO_WP : E_SEQ_PROCESS
VAR_INPUT
END_VAR
VAR
	ActiveSeq: STRING;
END_VAR
VAR
	
END_VAR
//THIS^._m_GeneralStepSetting(StepType:=E_STEP_STATE_TYPE.INIT,
ActiveSeq := TO_STRING(THIS^.eSeq);

CASE THIS^.stSeqCtrlGeneral.eActiveSeqState OF
E_SEQ_GENERAL.READY:;

	
E_SEQ_GENERAL.EXECUTE:;
	IF TRUE
	THEN
    THIS^.bRegulationTrigger := FALSE;
    THIS^.bPressureRegulationTrigger := FALSE;
		THIS^.stSeqCtrlGeneral.eActiveSeqState := E_SEQ_GENERAL.RESET;
	END_IF
  
E_SEQ_GENERAL.RESET:;
	stSeqCtrlGeneral.iInternalSeqStateCase := 0;
	IF TRUE
	THEN
		THIS^.stSeqCtrlGeneral.eActiveSeqState := E_SEQ_GENERAL.BUSY;
	END_IF
  
E_SEQ_GENERAL.BUSY:;
	CASE THIS^.stSeqCtrlGeneral.iInternalSeqStateCase OF
		0:	// Set work pressure
      IF TRUE
      AND THIS^.itfValve_PressureLimit.M_SetLimit(ePressureType:= E_PRESSURE_TYPE.VALUE, rLimit:= TO_REAL(THIS^.iTargetPressureAsValueA))
			THEN 
        THIS^.stSeqCtrlGeneral.iInternalSeqStateCase := 10;
			END_IF

    10:	// Switch on lock A valve
      IF TRUE
      AND THIS^.itfValve_LockA.M_ToWP1(tDelay:= T#0MS)
			THEN 
        IF THIS^.bDoableActing THEN
				  THIS^.stSeqCtrlGeneral.iInternalSeqStateCase := 20;
        ELSE
          THIS^.stSeqCtrlGeneral.iInternalSeqStateCase := 30;
        END_IF
			END_IF
      
    20:	// Switch on lock B valve
      IF TRUE
      AND THIS^.itfValve_LockB.M_ToWP1(tDelay:= T#0MS)
			THEN 
				THIS^.stSeqCtrlGeneral.iInternalSeqStateCase := 30;
			END_IF
      
    30:	// Set valve control
      IF TRUE
      AND THIS^.itfValve_CylCtrl.M_ValveCtrl(rSpeedInPercent:= THIS^.rSpeedInPercentToSet, tDelay:= T#0MS)
			THEN 
				THIS^.stSeqCtrlGeneral.iInternalSeqStateCase := 1000;
			END_IF
      
    1000: // Exit step
      IF TRUE
			THEN 
				THIS^.stSeqCtrlGeneral.iInternalSeqStateCase := 9999;
			END_IF
      
	ELSE
		THIS^.stSeqCtrlGeneral.eActiveSeqState := E_SEQ_GENERAL.DONE;  
	END_CASE
	THIS^.stSeqCtrlGeneral.strExtraInfo := CONCAT('Internal state: ', TO_STRING(THIS^.stSeqCtrlGeneral.iInternalSeqStateCase));

E_SEQ_GENERAL.DONE:;
  THIS^.bRegulationTrigger := THIS^.bRegulation;
  THIS^.bPressureRegulationTrigger := THIS^.bPressureRegulation;
  
E_SEQ_GENERAL.ERROR:;

E_SEQ_GENERAL.TIME_OUT:; 
IF TRUE
AND THIS^.stSeqCtrlGeneral.bTimeOutActiveQuit 
THEN
  THIS^.stSeqCtrlGeneral.strExtraInfo := 'Bitte quittieren und erneut testen';
  IF TRUE
  //AND itfOpMode.P_QUIT
  THEN
    THIS^.stSeqCtrlGeneral.eActiveSeqState := E_SEQ_GENERAL.EXECUTE;
	END_IF
  
END_IF

ELSE
  THIS^.stSeqCtrlGeneral.eActiveSeqState := E_SEQ_GENERAL.ERROR;
END_CASE
END_METHOD

METHOD PRIVATE _m_SequenceManager
VAR_INPUT
END_VAR
IF FALSE
//AND THIS^.eActiveSeqState=DONE 
AND eLastSeq<>eSeq
THEN
	IF THIS^.stSeqCtrlGeneral.eActiveSeqState<>E_SEQ_GENERAL.EXECUTE THEN
		THIS^.stSeqCtrlGeneral.eActiveSeqState:=E_SEQ_GENERAL.READY;
	END_IF
END_IF

eSeq := eNextSeq;

//DelayTimer und TimeOut Timer verwalten
stSeqCtrlGeneral.bActiveStep:=	TRUE
				AND eLastSeq					=	eSeq
				AND stSeqCtrlGeneral.eLastActiveSeqState			=	stSeqCtrlGeneral.eActiveSeqState
				AND	stSeqCtrlGeneral.iLastInternalSeqStateCase	=	stSeqCtrlGeneral.iInternalSeqStateCase
				;
			
IF NOT stSeqCtrlGeneral.bActiveStep THEN
	stSeqCtrlGeneral.bDelayActive:=FALSE;
	stSeqCtrlGeneral.bTimeOutActiveQuit:=FALSE;
	stSeqCtrlGeneral.bTimeOutActiveNoQuit:=FALSE;
  THIS^.stSeqCtrlGeneral.strExtraInfo:='';
END_IF

_m_SaveLastStep();
stSeqCtrlGeneral.tonDelay	(IN:=stSeqCtrlGeneral.bActiveStep AND stSeqCtrlGeneral.bDelayActive, 		PT:=stSeqCtrlGeneral.tDelay);
stSeqCtrlGeneral.tonTimeOut	(IN:=stSeqCtrlGeneral.bActiveStep AND (stSeqCtrlGeneral.bTimeOutActiveNoQuit OR stSeqCtrlGeneral.bTimeOutActiveQuit), 	PT:=stSeqCtrlGeneral.tTimeOut);
stSeqCtrlGeneral.tonStepTime	(IN:= stSeqCtrlGeneral.bActiveStep, PT:= T#24H);

IF stSeqCtrlGeneral.tonTimeOut.Q  THEN
	stSeqCtrlGeneral.eActiveSeqState:=E_SEQ_GENERAL.TIME_OUT;
END_IF

IF stSeqCtrlGeneral.iError<>0 THEN
	eSeq:=E_SEQ_CYLINDER.ERROR_SEQ;
END_IF



eLastSeq					:=	eSeq;
stSeqCtrlGeneral.eLastActiveSeqState			:=	stSeqCtrlGeneral.eActiveSeqState;
stSeqCtrlGeneral.iLastInternalSeqStateCase	:=	stSeqCtrlGeneral.iInternalSeqStateCase;

// Reset set ready state
IF THIS^.stSeqCtrlGeneral.bExitSetReadyState THEN
  THIS^.stSeqCtrlGeneral.bExitSetReadyState := FALSE;
END_IF
END_METHOD

(******************Description****************)
// This function allows variable speed control
(*********************************************)
METHOD PRIVATE _m_SpeedRegulation : BOOL
VAR_INPUT
END_VAR
IF TRUE
AND THIS^.rCurrentSpeedInMmPerS < THIS^.rSpeedInMmPerSToSet 
AND THIS^.rCorrectedSpeedPercent < 100
AND THIS^.bRegulationTrigger
AND NOT THIS^.bRegulationBusy
THEN
  IF ABS(THIS^.rCurrentSpeedInMmPerS - THIS^.rSpeedInMmPerSToSet) > 1 THEN
    //THIS^.rCorrectedSpeedPercent := THIS^.rCorrectedSpeedPercent + 0.25;
    THIS^.rCorrectedSpeedPercent := THIS^.rCorrectedSpeedPercent + ABS((THIS^.rCurrentSpeedInMmPerS - THIS^.rSpeedInMmPerSToSet) * THIS^.rSpeedRegulationFactor);
    THIS^.bCorrectionTrigger := TRUE;
  END_IF
ELSIF TRUE
AND THIS^.rCurrentSpeedInMmPerS > THIS^.rSpeedInMmPerSToSet 
AND THIS^.rCorrectedSpeedPercent > -100
AND THIS^.bRegulationTrigger
AND NOT THIS^.bRegulationBusy
THEN
  IF ABS(THIS^.rCurrentSpeedInMmPerS - THIS^.rSpeedInMmPerSToSet) > 1 THEN
    //THIS^.rCorrectedSpeedPercent := THIS^.rCorrectedSpeedPercent - 0.25;
    THIS^.rCorrectedSpeedPercent := THIS^.rCorrectedSpeedPercent - ABS((THIS^.rCurrentSpeedInMmPerS - THIS^.rSpeedInMmPerSToSet) * THIS^.rSpeedRegulationFactor);
    THIS^.bCorrectionTrigger := TRUE;
  END_IF
END_IF

// Valve value correction
IF THIS^.bCorrectionTrigger THEN
  THIS^.bRegulationBusy:= TRUE;
  CASE THIS^.uiRegulationSeq OF
    0:;
      IF THIS^.itfValve_CylCtrl.M_SetReady() THEN
        THIS^.uiRegulationSeq := 1;
	    END_IF
    1:;
      IF THIS^.itfValve_CylCtrl.M_ValveCtrl(rSpeedInPercent:= THIS^.rCorrectedSpeedPercent, tDelay:= T#0MS) THEN
        THIS^.bCorrectionTrigger := FALSE;
        THIS^.bRegulationBusy := FALSE;
        THIS^.uiRegulationSeq := 0;
	    END_IF
	END_CASE
END_IF
END_METHOD

METHOD PRIVATE _m_TimeOut : BOOL
VAR_INPUT
	bTimeoutActiveToQuit:	BOOL;
	bTimeOutActiveNoQuit:	BOOL;
	tTimeOut:				TIME;	
END_VAR
THIS^.stSeqCtrlGeneral.bTimeOutActiveQuit:=	bTimeoutActiveToQuit;
THIS^.stSeqCtrlGeneral.bTimeOutActiveNoQuit:=	bTimeOutActiveNoQuit;
THIS^.stSeqCtrlGeneral.tTimeOut:=			tTimeOut;
_m_TimeOut:=FALSE;
IF THIS^.stSeqCtrlGeneral.tonTimeOut.Q THEN
	_m_TimeOut:=TRUE;
END_IF
END_METHOD

METHOD FB_init : BOOL
VAR_INPUT
	bInitRetains : BOOL; // if TRUE, the retain variables are initialized (warm start / cold start)
	bInCopyCode : BOOL;  // if TRUE, the instance afterwards gets moved into the copy code (online change)
  
  itfLogEvents: 										                      I_HANDLE_EVENTS;
  itfOpMode:											                        I_OP_MODE;
  itfOpModeVisu:											                    I_OP_MODE_PAUSE_VISU;
  itfValve_CylCtrl:                                       I_VALVE_X_3_PROP;
  itfValve_LockA:                                         I_VALVE_X_2;
  itfValve_LockB:                                         I_VALVE_X_2;
  itfValve_PressureLimit:                                 I_PRV_PROP; 
  rEndPosTol:                                             REAL;
  /// Volume flow in l/min or dm³/min
  rPumpVolumeFlow:                                        REAL; // Volumenstrom
  /// Pump efficiency factor (0,5-1)
  rPumpEfficiencyFactor:                                  REAL; // Wirkungsgrad
END_VAR
THIS^.itfLogEvents := itfLogEvents;
THIS^.itfOpMode := itfOpMode;
THIS^.itfOpModeVisu := itfOpModeVisu;
THIS^.itfValve_CylCtrl := itfValve_CylCtrl;
THIS^.itfValve_LockA := itfValve_LockA;
THIS^.itfValve_LockB := itfValve_LockB;
THIS^.itfValve_PressureLimit := itfValve_PressureLimit;
THIS^.rEndPosTol := rEndPosTol;
THIS^.rPumpVolumeFlow := rPumpVolumeFlow;
THIS^.rPumpEfficiencyFactor := rPumpEfficiencyFactor;
END_METHOD

METHOD M_OpenLockValves : BOOL
VAR_INPUT
	bOpenChA	: BOOL;
	bOpenChB	: BOOL;
END_VAR
M_OpenLockValves := THIS^.stSeqCtrlGeneral.eActiveSeqState = E_SEQ_GENERAL.DONE;

// Assign input
THIS^.bOpenChA := bOpenChA;
THIS^.bOpenChB := bOpenChB;

// General
IF THIS^.stSeqCtrlGeneral.eActiveSeqState = E_SEQ_GENERAL.READY THEN
  THIS^.eNextSeq := E_SEQ_CYLINDER.OPEN_LOCK_VALVES;
  THIS^.stSeqCtrlGeneral.eActiveSeqState := E_SEQ_GENERAL.EXECUTE;
END_IF
END_METHOD

METHOD M_PressureCalibration : BOOL
M_PressureCalibration := THIS^.stSeqCtrlGeneral.eActiveSeqState = E_SEQ_GENERAL.DONE;

// Assign input

// General
IF THIS^.stSeqCtrlGeneral.eActiveSeqState = E_SEQ_GENERAL.READY THEN
  THIS^.eNextSeq := E_SEQ_CYLINDER.PRESSURE_CALIBRATION;
  THIS^.stSeqCtrlGeneral.eActiveSeqState := E_SEQ_GENERAL.EXECUTE;
END_IF
END_METHOD

METHOD M_Reset : BOOL
M_Reset := THIS^.stSeqCtrlGeneral.eActiveSeqState = E_SEQ_GENERAL.DONE;

// General
IF THIS^.stSeqCtrlGeneral.eActiveSeqState = E_SEQ_GENERAL.READY THEN
  THIS^.eNextSeq := E_SEQ_CYLINDER.INIT;
  THIS^.stSeqCtrlGeneral.eActiveSeqState := E_SEQ_GENERAL.EXECUTE;
END_IF
END_METHOD

{warning 'Methodenimplementierung hinzufügen'}
(*=== Method: M_Run  ============================================

 @brief: Here is the global code (Timer, Event, Flange,...)*)
METHOD M_Run
END_METHOD

METHOD M_SetMaxPos : BOOL
M_SetMaxPos := THIS^.stSeqCtrlGeneral.eActiveSeqState = E_SEQ_GENERAL.DONE;

// General
IF THIS^.stSeqCtrlGeneral.eActiveSeqState = E_SEQ_GENERAL.READY THEN
  THIS^.eNextSeq := E_SEQ_CYLINDER.SET_MAX_POS;
  THIS^.stSeqCtrlGeneral.eActiveSeqState := E_SEQ_GENERAL.EXECUTE;
END_IF
END_METHOD

METHOD M_SetReady : BOOL
VAR_INPUT
END_VAR
M_SetReady := stSeqCtrlGeneral.eActiveSeqState = E_SEQ_GENERAL.READY;

THIS^.stSeqCtrlGeneral.eActiveSeqState := E_SEQ_GENERAL.READY;
END_METHOD

METHOD M_SetWorkPressure : BOOL
VAR_INPUT
  ePressureType:                   E_PRESSURE_TYPE;
  rWorkPressure:                   REAL;
END_VAR
M_SetWorkPressure := THIS^.stSeqCtrlGeneral.eActiveSeqState = E_SEQ_GENERAL.DONE;

// Assign input
IF ePressureType = E_PRESSURE_TYPE.BAR THEN
  THIS^.rTargetPressureInBarA := THIS^.rTargetPressureInBarB := rWorkPressure;
  THIS^.rTargetPressureInForceA := rWorkPressure / 10 * THIS^.lrPistonSurfaceA;
  THIS^.rTargetPressureInForceB := rWorkPressure / 10 * THIS^.lrPistonSurfaceB;
  THIS^.rTargetPressureInPercentA := THIS^.rTargetPressureInPercentB := 100 / THIS^.itfValve_PressureLimit.P_MaxLimitInBar * rWorkPressure;
  THIS^.iTargetPressureAsValueA := THIS^.iTargetPressureAsValueB := TO_INT(F_InterpolLinear(lrValueUnscale := rWorkPressure , arrCalibrate:= listCylCalibration, iPts:= 7));
ELSIF ePressureType = E_PRESSURE_TYPE.FORCE THEN
  THIS^.rTargetPressureInForceA := THIS^.rTargetPressureInForceB := rWorkPressure;;
  THIS^.rTargetPressureInBarA := THIS^.rTargetPressureInForceA / THIS^.lrPistonSurfaceA * 10;
  THIS^.rTargetPressureInBarB := THIS^.rTargetPressureInForceB / THIS^.lrPistonSurfaceB * 10;
  THIS^.rTargetPressureInPercentA := 100 / THIS^.itfValve_PressureLimit.P_MaxLimitInBar * THIS^.rTargetPressureInBarA;
  THIS^.rTargetPressureInPercentB := 100 / THIS^.itfValve_PressureLimit.P_MaxLimitInBar * THIS^.rTargetPressureInBarB;
  THIS^.iTargetPressureAsValueA := TO_INT(F_InterpolLinear(lrValueUnscale := THIS^.rTargetPressureInBarA , arrCalibrate:= listCylCalibration, iPts:= 7));
  THIS^.iTargetPressureAsValueB := TO_INT(F_InterpolLinear(lrValueUnscale := THIS^.rTargetPressureInBarB , arrCalibrate:= listCylCalibration, iPts:= 7));
ELSIF ePressureType = E_PRESSURE_TYPE.PERCENT THEN
  THIS^.rTargetPressureInPercentA := THIS^.rTargetPressureInPercentB := rWorkPressure;
  THIS^.rTargetPressureInBarA := THIS^.rTargetPressureInBarB := THIS^.itfValve_PressureLimit.P_MaxLimitInBar / 100 * rWorkPressure;
  THIS^.rTargetPressureInForceA := THIS^.rTargetPressureInBarA / 10 * THIS^.lrPistonSurfaceA;
  THIS^.rTargetPressureInForceB := THIS^.rTargetPressureInBarB / 10 * THIS^.lrPistonSurfaceB;
  THIS^.iTargetPressureAsValueA := TO_INT(F_InterpolLinear(lrValueUnscale := THIS^.rTargetPressureInBarA , arrCalibrate:= listCylCalibration, iPts:= 7));
  THIS^.iTargetPressureAsValueB := TO_INT(F_InterpolLinear(lrValueUnscale := THIS^.rTargetPressureInBarB , arrCalibrate:= listCylCalibration, iPts:= 7));
ELSE
  THIS^.iTargetPressureAsValueA := THIS^.iTargetPressureAsValueB := TO_INT(rWorkPressure);
END_IF

// General
IF THIS^.stSeqCtrlGeneral.eActiveSeqState = E_SEQ_GENERAL.READY THEN
  THIS^.eNextSeq := E_SEQ_CYLINDER.SET_WORK_PRESSURE;
  THIS^.stSeqCtrlGeneral.eActiveSeqState := E_SEQ_GENERAL.EXECUTE;
END_IF
END_METHOD

METHOD M_SetZeroPos : BOOL
M_SetZeroPos := THIS^.stSeqCtrlGeneral.eActiveSeqState = E_SEQ_GENERAL.DONE;

// General
IF THIS^.stSeqCtrlGeneral.eActiveSeqState = E_SEQ_GENERAL.READY THEN
  THIS^.eNextSeq := E_SEQ_CYLINDER.SET_ZERO_POS;
  THIS^.stSeqCtrlGeneral.eActiveSeqState := E_SEQ_GENERAL.EXECUTE;
END_IF
END_METHOD

METHOD M_Stop : BOOL
M_Stop := THIS^.stSeqCtrlGeneral.eActiveSeqState = E_SEQ_GENERAL.DONE;

// Assign input
THIS^.bRegulation := FALSE;
THIS^.rSpeedInMmPerSToSet := 0;
THIS^.rSpeedInPercentToSet := 0;
THIS^.rCorrectedSpeedPercent := 0;
THIS^.bPressureRegulation := FALSE;
THIS^.rActiveForce := 0;
THIS^.iCorrectedPressureAsValue := 0;
THIS^.bPressureRegulationTrigger := FALSE;
THIS^.bPressureRegulationBusy := FALSE;
THIS^.bPressureCorrectionTrigger := FALSE;

// General
IF THIS^.stSeqCtrlGeneral.eActiveSeqState = E_SEQ_GENERAL.READY THEN
  THIS^.eNextSeq := E_SEQ_CYLINDER.STOP;
  THIS^.stSeqCtrlGeneral.eActiveSeqState := E_SEQ_GENERAL.EXECUTE;
END_IF
END_METHOD

METHOD M_StopAndLock : BOOL
M_StopAndLock := THIS^.stSeqCtrlGeneral.eActiveSeqState = E_SEQ_GENERAL.DONE;

// Assign input
THIS^.bRegulation := FALSE;
THIS^.rSpeedInMmPerSToSet := 0;
THIS^.rSpeedInPercentToSet := 0;
THIS^.rCorrectedSpeedPercent := 0;
THIS^.bPressureRegulation := FALSE;
THIS^.rActiveForce := 0;
THIS^.iCorrectedPressureAsValue := 0;
THIS^.bPressureRegulationTrigger := FALSE;
THIS^.bPressureRegulationBusy := FALSE;
THIS^.bPressureCorrectionTrigger := FALSE;

// General
IF THIS^.stSeqCtrlGeneral.eActiveSeqState = E_SEQ_GENERAL.READY THEN
  THIS^.eNextSeq := E_SEQ_CYLINDER.STOP_AND_LOCK;
  THIS^.stSeqCtrlGeneral.eActiveSeqState := E_SEQ_GENERAL.EXECUTE;
END_IF
END_METHOD

METHOD M_ToHP : BOOL
VAR_INPUT
  /// Bar | Force in N | Percent 0-100 | Value 0-32767
  ePressureType:            E_PRESSURE_TYPE;
  rWorkPressure:            REAL;
  /// Just need for prop valve
  eSpeedType:               E_SPEED_TYPE;
  rSpeed:                   REAL;
END_VAR
VAR
  
END_VAR
M_ToHP := THIS^.stSeqCtrlGeneral.eActiveSeqState = E_SEQ_GENERAL.DONE;

// Der prozentualler Wert wurde pauschal um -15 verringert, da sonst die automatische Regullierung zuviel nachregeln muss (Toter Ventilbereich).
// Hier mit weiteren Varianten testen, wie sich die Regelung verhällt, evtl parametrierbar.

// Assign input
IF eSpeedType = E_SPEED_TYPE.MM_PER_SECOND THEN
  THIS^.bRegulation := TRUE;
  THIS^.rSpeedInMmPerSToSet := -ABS(rSpeed);
  THIS^.rSpeedInPercentToSet := THIS^.rCorrectedSpeedPercent := -15(*-ABS((3 * THIS^.lrPistonSurfaceB * THIS^.rPumpEfficiencyFactor * rSpeed) / (500 * THIS^.rPumpVolumeFlow))*);
ELSE
  THIS^.bRegulation := FALSE;
  THIS^.rSpeedInPercentToSet := THIS^.rCorrectedSpeedPercent := -ABS(rSpeed);
END_IF
IF THIS^.rSpeedInPercentToSet < -100 THEN
  THIS^.rSpeedInPercentToSet := THIS^.rCorrectedSpeedPercent := -100;
END_IF

IF ePressureType = E_PRESSURE_TYPE.BAR THEN
  THIS^.rTargetPressureInBarA := THIS^.rTargetPressureInBarB := rWorkPressure;
  THIS^.rTargetPressureInForceA := rWorkPressure / 10 * THIS^.lrPistonSurfaceA;
  THIS^.rTargetPressureInForceB := rWorkPressure / 10 * THIS^.lrPistonSurfaceB;
  THIS^.rTargetPressureInPercentA := THIS^.rTargetPressureInPercentB := 100 / THIS^.itfValve_PressureLimit.P_MaxLimitInBar * rWorkPressure;
  THIS^.iTargetPressureAsValueA := THIS^.iTargetPressureAsValueB := THIS^.iCorrectedPressureAsValue := TO_INT(F_InterpolLinear(lrValueUnscale := rWorkPressure , arrCalibrate:= listCylCalibration, iPts:= 7));
ELSIF ePressureType = E_PRESSURE_TYPE.FORCE THEN
  THIS^.rTargetPressureInForceA := THIS^.rTargetPressureInForceB := rWorkPressure;;
  THIS^.rTargetPressureInBarA := THIS^.rTargetPressureInForceA / THIS^.lrPistonSurfaceA * 10;
  THIS^.rTargetPressureInBarB := THIS^.rTargetPressureInForceB / THIS^.lrPistonSurfaceB * 10;
  THIS^.rTargetPressureInPercentA := 100 / THIS^.itfValve_PressureLimit.P_MaxLimitInBar * THIS^.rTargetPressureInBarA;
  THIS^.rTargetPressureInPercentB := 100 / THIS^.itfValve_PressureLimit.P_MaxLimitInBar * THIS^.rTargetPressureInBarB;
  THIS^.iTargetPressureAsValueA := THIS^.iCorrectedPressureAsValue := TO_INT(F_InterpolLinear(lrValueUnscale := THIS^.rTargetPressureInBarA , arrCalibrate:= listCylCalibration, iPts:= 7));
  THIS^.iTargetPressureAsValueB := TO_INT(F_InterpolLinear(lrValueUnscale := THIS^.rTargetPressureInBarB , arrCalibrate:= listCylCalibration, iPts:= 7));
ELSIF ePressureType = E_PRESSURE_TYPE.PERCENT THEN
  THIS^.rTargetPressureInPercentA := THIS^.rTargetPressureInPercentB := rWorkPressure;
  THIS^.rTargetPressureInBarA := THIS^.rTargetPressureInBarB := THIS^.itfValve_PressureLimit.P_MaxLimitInBar / 100 * rWorkPressure;
  THIS^.rTargetPressureInForceA := THIS^.rTargetPressureInBarA / 10 * THIS^.lrPistonSurfaceA;
  THIS^.rTargetPressureInForceB := THIS^.rTargetPressureInBarB / 10 * THIS^.lrPistonSurfaceB;
  THIS^.iTargetPressureAsValueA := THIS^.iCorrectedPressureAsValue := TO_INT(F_InterpolLinear(lrValueUnscale := THIS^.rTargetPressureInBarA , arrCalibrate:= listCylCalibration, iPts:= 7));
  THIS^.iTargetPressureAsValueB := TO_INT(F_InterpolLinear(lrValueUnscale := THIS^.rTargetPressureInBarB , arrCalibrate:= listCylCalibration, iPts:= 7));
ELSE
  THIS^.iTargetPressureAsValueA := THIS^.iTargetPressureAsValueB := THIS^.iCorrectedPressureAsValue := TO_INT(rWorkPressure);
END_IF
THIS^.bPressureRegulation := TRUE;

// General
IF THIS^.stSeqCtrlGeneral.eActiveSeqState = E_SEQ_GENERAL.READY THEN
  THIS^.eNextSeq := E_SEQ_CYLINDER.TO_HP;
  THIS^.stSeqCtrlGeneral.eActiveSeqState := E_SEQ_GENERAL.EXECUTE;
END_IF
END_METHOD

METHOD M_ToSetPos : BOOL
VAR_INPUT
  lrToSetPos:                 LREAL;
  /// Just need for prop valve
  eSpeedType:               E_SPEED_TYPE;
  rSpeed:                   REAL; 
END_VAR
VAR
  lrCylPistonSurface:       LREAL;
END_VAR
M_ToSetPos := THIS^.stSeqCtrlGeneral.eActiveSeqState = E_SEQ_GENERAL.DONE;

// Assign input
THIS^.lrToSetPos := lrToSetPos;
IF eSpeedType = E_SPEED_TYPE.MM_PER_SECOND THEN
  THIS^.rSpeedInMmPerSToSet := rSpeed;
  // Convert mm/s to percent
  IF THIS^.lrPos < lrToSetPos THEN
    lrCylPistonSurface := THIS^.lrPistonSurfaceA;
  ELSE
    lrCylPistonSurface := THIS^.lrPistonSurfaceB;
  END_IF
  THIS^.rSpeedInPercentToSet := ABS((3 * lrCylPistonSurface * THIS^.rPumpEfficiencyFactor * rSpeed) / (500 * THIS^.rPumpVolumeFlow));
ELSE
  THIS^.rSpeedInPercentToSet := ABS(rSpeed);
END_IF
IF THIS^.rSpeedInPercentToSet > 100 THEN
  THIS^.rSpeedInPercentToSet := 100;
END_IF

// General
IF THIS^.stSeqCtrlGeneral.eActiveSeqState = E_SEQ_GENERAL.READY THEN
  THIS^.eNextSeq := E_SEQ_CYLINDER.TO_SET_POS;
  THIS^.stSeqCtrlGeneral.eActiveSeqState := E_SEQ_GENERAL.EXECUTE;
END_IF
END_METHOD

METHOD M_ToWP : BOOL
VAR_INPUT
  /// Bar | Force in N | Percent 0-100 | Value 0-32767
  ePressureType:            E_PRESSURE_TYPE;
  rWorkPressure:            REAL;
  /// Just need for prop valve
  eSpeedType:               E_SPEED_TYPE;
  rSpeed:                   REAL;
END_VAR
M_ToWP := THIS^.stSeqCtrlGeneral.eActiveSeqState = E_SEQ_GENERAL.DONE;

// Der prozentualler Wert wurde pauschal um -5 verringert, da sonst die automatische Regullierung zuviel nachregeln muss (Toter Ventilbereich).
// Hier mit weiteren Varianten testen, wie sich die Regelung verhällt, evtl parametrierbar.

// Assign input
IF eSpeedType = E_SPEED_TYPE.MM_PER_SECOND THEN
  THIS^.bRegulation := TRUE;
  THIS^.rSpeedInMmPerSToSet := ABS(rSpeed);
  THIS^.rSpeedInPercentToSet := THIS^.rCorrectedSpeedPercent := 15(*ABS((3 * THIS^.lrPistonSurfaceA * THIS^.rPumpEfficiencyFactor * rSpeed) / (500 * THIS^.rPumpVolumeFlow))*);
ELSE
  THIS^.bRegulation := FALSE;
  THIS^.rSpeedInPercentToSet := THIS^.rCorrectedSpeedPercent := ABS(rSpeed);
END_IF
IF THIS^.rSpeedInPercentToSet > 100 THEN
  THIS^.rSpeedInPercentToSet := THIS^.rCorrectedSpeedPercent := 100;
END_IF

IF ePressureType = E_PRESSURE_TYPE.BAR THEN
  THIS^.rTargetPressureInBarA := THIS^.rTargetPressureInBarB := rWorkPressure;
  THIS^.rTargetPressureInForceA := rWorkPressure / 10 * THIS^.lrPistonSurfaceA;
  THIS^.rTargetPressureInForceB := rWorkPressure / 10 * THIS^.lrPistonSurfaceB;
  THIS^.rTargetPressureInPercentA := THIS^.rTargetPressureInPercentB := 100 / THIS^.itfValve_PressureLimit.P_MaxLimitInBar * rWorkPressure;
  THIS^.iTargetPressureAsValueA := THIS^.iTargetPressureAsValueB := THIS^.iCorrectedPressureAsValue := TO_INT(F_InterpolLinear(lrValueUnscale := rWorkPressure , arrCalibrate:= listCylCalibration, iPts:= 7));
ELSIF ePressureType = E_PRESSURE_TYPE.FORCE THEN
  THIS^.rTargetPressureInForceA := THIS^.rTargetPressureInForceB := rWorkPressure;;
  THIS^.rTargetPressureInBarA := THIS^.rTargetPressureInForceA / THIS^.lrPistonSurfaceA * 10;
  THIS^.rTargetPressureInBarB := THIS^.rTargetPressureInForceB / THIS^.lrPistonSurfaceB * 10;
  THIS^.rTargetPressureInPercentA := 100 / THIS^.itfValve_PressureLimit.P_MaxLimitInBar * THIS^.rTargetPressureInBarA;
  THIS^.rTargetPressureInPercentB := 100 / THIS^.itfValve_PressureLimit.P_MaxLimitInBar * THIS^.rTargetPressureInBarB;
  THIS^.iTargetPressureAsValueA := THIS^.iCorrectedPressureAsValue := TO_INT(F_InterpolLinear(lrValueUnscale := THIS^.rTargetPressureInBarA , arrCalibrate:= listCylCalibration, iPts:= 7));
  THIS^.iTargetPressureAsValueB := TO_INT(F_InterpolLinear(lrValueUnscale := THIS^.rTargetPressureInBarB , arrCalibrate:= listCylCalibration, iPts:= 7));
ELSIF ePressureType = E_PRESSURE_TYPE.PERCENT THEN
  THIS^.rTargetPressureInPercentA := THIS^.rTargetPressureInPercentB := rWorkPressure;
  THIS^.rTargetPressureInBarA := THIS^.rTargetPressureInBarB := THIS^.itfValve_PressureLimit.P_MaxLimitInBar / 100 * rWorkPressure;
  THIS^.rTargetPressureInForceA := THIS^.rTargetPressureInBarA / 10 * THIS^.lrPistonSurfaceA;
  THIS^.rTargetPressureInForceB := THIS^.rTargetPressureInBarB / 10 * THIS^.lrPistonSurfaceB;
  THIS^.iTargetPressureAsValueA := THIS^.iCorrectedPressureAsValue := TO_INT(F_InterpolLinear(lrValueUnscale := THIS^.rTargetPressureInBarA , arrCalibrate:= listCylCalibration, iPts:= 7));
  THIS^.iTargetPressureAsValueB := TO_INT(F_InterpolLinear(lrValueUnscale := THIS^.rTargetPressureInBarB , arrCalibrate:= listCylCalibration, iPts:= 7));
ELSE
  THIS^.iTargetPressureAsValueA := THIS^.iTargetPressureAsValueB := THIS^.iCorrectedPressureAsValue := TO_INT(rWorkPressure);
END_IF
THIS^.bPressureRegulation := TRUE;

// General
IF THIS^.stSeqCtrlGeneral.eActiveSeqState = E_SEQ_GENERAL.READY THEN
  THIS^.eNextSeq := E_SEQ_CYLINDER.TO_WP;
  THIS^.stSeqCtrlGeneral.eActiveSeqState := E_SEQ_GENERAL.EXECUTE;
END_IF
END_METHOD

PROPERTY P_ActiveDirection : STRING
GET
IF THIS^.itfValve_CylCtrl.P_CurrentVal < - 100 THEN
  P_ActiveDirection := 'Moove to home position';
ELSIF THIS^.itfValve_CylCtrl.P_CurrentVal > 100 THEN
  P_ActiveDirection := 'Moove to work position';
ELSE
  P_ActiveDirection := 'Stop';
END_IF
END_GET
END_PROPERTY

{warning 'Eigenschaftenimplementierung hinzufügen'}
PROPERTY P_CurrentForceInKN : REAL
GET
IF THIS^.rCorrectedSpeedPercent > 0 THEN
  P_CurrentForceInKN := THIS^.rCurrentPressureInBar / 10000 * THIS^.lrPistonSurfaceA;
  THIS^.rActiveForce := THIS^.rTargetPressureInForceA;
ELSE
  P_CurrentForceInKN := THIS^.rCurrentPressureInBar / 10000 * THIS^.lrPistonSurfaceB;
  THIS^.rActiveForce := THIS^.rTargetPressureInForceB;
END_IF
END_GET
END_PROPERTY

{warning 'Eigenschaftenimplementierung hinzufügen'}
PROPERTY P_DoubleActing : BOOL
GET
P_DoubleActing := THIS^.bDoableActing;
END_GET
END_PROPERTY

{warning 'Eigenschaftenimplementierung hinzufügen'}
(*=== Property: P_Event  ============================================

 @param [set]: 	Set the Structure "ST_EVENT" from another Object
 @param [get]: 	Return the Structure "ST_EVENT", it contains the actual 
					event of the Object *)
PROPERTY P_Event : GenLib.ST_EVENT
GET
END_GET
SET
END_SET
END_PROPERTY

{warning 'Eigenschaftenimplementierung hinzufügen'}
(*=== Property: P_FullObjectPath  ============================================

 @param [set]: 	Set the Object Path (Clear String of Object)
 @param [get]: 	Return the Objectpath *)
PROPERTY P_FullObjectPath : STRING
GET
P_FullObjectPath := strInstancePath;
END_GET
SET
strInstancePath := P_FullObjectPath;
END_SET
END_PROPERTY

{warning 'Eigenschaftenimplementierung hinzufügen'}
(*=== Property: P_Global_Ack  ============================================

 @param [set]: 	Set the Bit for Ack from another Object
 @param [get]: 	Return the state of Ack Bit*)
PROPERTY P_Global_Ack : BOOL
GET
END_GET
SET
END_SET
END_PROPERTY

{warning 'Eigenschaftenimplementierung hinzufügen'}
(*=== Property: P_GlobalID  ============================================

 @param [set]: 	-
 @param [get]: 	Return the string of instance path*)
PROPERTY P_GlobalID : STRING
GET
END_GET
END_PROPERTY

{warning 'Eigenschaftenimplementierung hinzufügen'}
PROPERTY P_MaxPosVal : LREAL
GET
P_MaxPosVal := THIS^.lrPosMax;
END_GET
END_PROPERTY

{warning 'Eigenschaftenimplementierung hinzufügen'}
PROPERTY P_MinPosVal : LREAL
GET
P_MinPosVal := THIS^.lrPosZero;
END_GET
END_PROPERTY

{warning 'Eigenschaftenimplementierung hinzufügen'}
PROPERTY P_PistonSurfaceA : LREAL
GET
P_PistonSurfaceA := THIS^.lrPistonSurfaceA;
END_GET
END_PROPERTY

{warning 'Eigenschaftenimplementierung hinzufügen'}
PROPERTY P_PistonSurfaceB : LREAL
GET
P_PistonSurfaceB := THIS^.lrPistonSurfaceB;
END_GET
END_PROPERTY

PROPERTY P_Position : LREAL
GET
P_Position := THIS^.lrPos;
END_GET
END_PROPERTY

{warning 'Eigenschaftenimplementierung hinzufügen'}
PROPERTY P_PositionAbs : LREAL
GET
P_PositionAbs := THIS^.lrCurrentPosAbs / 1000;
END_GET
END_PROPERTY

{warning 'Eigenschaftenimplementierung hinzufügen'}
PROPERTY P_PressureChA : REAL
GET
P_PressureChA := THIS^.rCurrentPressureInBarA;
END_GET
END_PROPERTY

{warning 'Eigenschaftenimplementierung hinzufügen'}
PROPERTY P_PressureChB : REAL
GET
P_PressureChB := THIS^.rCurrentPressureInBarB;
END_GET
END_PROPERTY

{warning 'Eigenschaftenimplementierung hinzufügen'}
PROPERTY P_PressureOk : BOOL
GET
//P_PRessureOk := ABS(rSetPressure - P_WorkPressure) < rEndPosTol;
END_GET
END_PROPERTY

{warning 'Eigenschaftenimplementierung hinzufügen'}
PROPERTY P_ReadyState : BOOL
GET
P_ReadyState := THIS^.stSeqCtrlGeneral.eActiveSeqState = E_SEQ_GENERAL.READY;
END_GET
END_PROPERTY

PROPERTY P_SpeedInMmPerSecond : REAL
GET
P_SpeedInMmPerSecond := THIS^.rCurrentSpeedInMmPerS;
END_GET
END_PROPERTY

{warning 'Eigenschaftenimplementierung hinzufügen'}
PROPERTY P_SpeedInPercent : LREAL
GET
P_SpeedInPercent := THIS^.rSpeedInPercentToSet;
END_GET
END_PROPERTY

PROPERTY P_StrokeLength : REAL
GET
P_StrokeLength := THIS^.rStrokeLength;
END_GET
END_PROPERTY

{warning 'Eigenschaftenimplementierung hinzufügen'}
PROPERTY P_StrokeLengthInitialized : BOOL
GET
P_StrokeLengthInitialized := THIS^.bStrokeLengthInitialized;
END_GET
SET
THIS^.bStrokeLengthInitialized := P_StrokeLengthInitialized;
END_SET
END_PROPERTY

PROPERTY P_WorkPressure : REAL
GET
P_WorkPressure := THIS^.rCurrentPressureInBar;
END_GET
END_PROPERTY

END_FUNCTION_BLOCK

(* stored: Version 1.1.0.1, ProductVersion 3.1.4024.12
   POU FB_CYLINDER_DA_TESTDEV2_4: Id {97ea8e37-52c6-4c5b-b9f6-4c7c70082a8f}, SpecialFunc None
   Folder PRIVAT: Id {8e2f15c2-a514-4057-96f5-a6a18a5d19c5}
   Folder SEQUENCE: Id {9e86da35-320f-4ee3-8510-8e6cc04be184}
   Method _m_DebugManager: Id {79d2b68c-22b0-4cdf-bd60-071c4851d8b7}
   Method _m_Delay: Id {856feeca-3e3a-4609-8b25-ce1f35e7bb13}
   Method _m_GeneralStepSetting: Id {b50d0c35-3f23-44d1-a808-5e1c1c35d80d}
   Method _m_HMI: Id {1c279bcb-26eb-4900-8dde-ac5b0eb3a667}
   Method _m_ManualOperation: Id {59d66084-9529-430f-8e53-6a67aff100f7}
   Method _m_PressureCalibration: Id {a29df983-2563-417d-b988-6acbf555ea9d}
   Method _m_PressureRegulation: Id {c5939910-43d2-4b7a-9d0f-32050bbd5181}
   Method _m_Recording: Id {f191d7fb-3df2-400d-b56b-38bef0fcbe76}
   Method _m_SaveLastStep: Id {5cf31f0f-e3bf-48fa-9ae6-48ef078b02e3}
   Method _m_Seq_INIT: Id {0dbbe223-f4f7-4907-a129-a8f58878da9e}
   Method _m_Seq_OPEN_LOCK_VALVES: Id {fba68cf5-e454-4578-97e5-2876b03c4464}
   Method _m_Seq_PRESSURE_CALIBRATION: Id {66fdb8d7-8ea4-434e-934c-e1d9b08d5d90}
   Method _m_Seq_SET_MAX_POS: Id {1c313491-53e4-4cb6-b8c4-19c72d5e0c3f}
   Method _m_Seq_SET_WORK_PRESSURE: Id {5bd8dfdc-3e09-42da-9a69-5d1f7166ee39}
   Method _m_Seq_SET_ZERO_POS: Id {a68ba7e8-2e89-436b-979d-7848b42749a0}
   Method _m_Seq_STOP: Id {3f4cb39c-87c8-45d7-83f9-d788327f0fda}
   Method _m_Seq_STOP_AND_LOCK: Id {e676dac5-cdf7-4008-b679-850265bd659a}
   Method _m_Seq_TO_HP: Id {277af6aa-4d66-4668-9815-97a21a93fcb2}
   Method _m_Seq_TO_SET_POS: Id {089e07e1-50e6-4787-97f9-672766abf814}
   Method _m_Seq_TO_WP: Id {8abb5d2e-1ad0-4a09-baa5-337f73174c94}
   Method _m_SequenceManager: Id {e0143faa-af89-4598-bb90-50264b1e57a3}
   Method _m_SpeedRegulation: Id {390b7281-9df3-484d-b044-f5b31eb72aa5}
   Method _m_TimeOut: Id {c67cd674-c2eb-411d-97f5-102e7d764c60}
   Method FB_init: Id {2d7848a9-7666-4c1b-bdd6-8592fa49e770}
   Method M_OpenLockValves: Id {484cdb60-7628-41ea-9551-915c289f1d2c}
   Method M_PressureCalibration: Id {8539f8c3-9add-4de0-87fe-d2501e9b08af}
   Method M_Reset: Id {a2440b5a-844c-4787-8936-818037fdbc3a}
   Method M_Run: Id {bac08aef-62ee-42c7-be92-a71fb3d1a55d}
   Method M_SetMaxPos: Id {3bb6a456-81e1-4ef7-af7b-aa7c5409cce1}
   Method M_SetReady: Id {e041a2a1-c4ec-4a2c-a127-248b8d3b6def}
   Method M_SetWorkPressure: Id {0d7061f5-c55e-4e7d-bdb4-23fde1282b6d}
   Method M_SetZeroPos: Id {48938c9a-b8d2-4664-b23c-c019e6c4eb56}
   Method M_Stop: Id {31fdab29-7478-4d54-8099-8513d5f1cbbc}
   Method M_StopAndLock: Id {d4415774-5ea1-415c-8baa-883958f9c000}
   Method M_ToHP: Id {3c2757ed-86f0-4ed3-afbe-3e0746100c22}
   Method M_ToSetPos: Id {de2ad4a3-4a87-462d-957e-dd66f58826a0}
   Method M_ToWP: Id {f20fedb6-d99d-406d-8512-39518e1da757}
   Property P_ActiveDirection: Id {d1d63849-d280-4181-864f-ef6f2b0ba811}
   Get Get: Id {24ba67c3-5f38-41af-bd11-26b17c7f287b}
   Property P_CurrentForceInKN: Id {1d02f2e1-3409-4c3a-aaab-7f8ea3fd07ce}
   Get Get: Id {3e702893-cedd-422c-a252-5d8c5eeab856}
   Property P_DoubleActing: Id {e5d046bb-75a7-45bc-83b1-07bc7309f718}
   Get Get: Id {9ca19a63-b300-45f6-a6dd-9225e1394b17}
   Property P_Event: Id {30513b81-8bc3-49ee-bc61-4bd225b5e5b4}
   Get Get: Id {d4120ef9-cd8a-4717-919b-581a8982f3f6}
   Set Set: Id {2dcf4109-207b-4e9d-bf86-a576c4f29ce1}
   Property P_FullObjectPath: Id {968a1f43-57d4-4dd9-9f8a-4b71bfefb580}
   Get Get: Id {aa86b76d-fc32-48e6-9bbd-e298cd9002a5}
   Set Set: Id {02187ba3-5dc4-4e46-83f1-b8493e52ce49}
   Property P_Global_Ack: Id {d5149326-ed7b-4c18-8372-65df86598c2e}
   Get Get: Id {2113a43b-4ba7-4f6c-92d4-4175892496d8}
   Set Set: Id {6c6a82ae-8186-4435-8723-296c67333df8}
   Property P_GlobalID: Id {b048aa7e-5965-469e-a6bd-3352eea42d6c}
   Get Get: Id {d0e44e42-c828-44e5-bbc6-145dce7a0e2e}
   Property P_MaxPosVal: Id {6f779c1b-174d-4e29-9797-b01d37391d84}
   Get Get: Id {ce6e330b-5388-4a2a-8628-aa5048131cee}
   Property P_MinPosVal: Id {e8f350dc-ba59-42e4-bb87-e858560eb644}
   Get Get: Id {6193b7c8-a22d-4db1-87bf-8632876684c7}
   Property P_PistonSurfaceA: Id {b27a0bf9-1668-4ed4-883e-62f9b4aaa0ec}
   Get Get: Id {32b0d532-4f6b-42ad-a6eb-8fbdb5cd00ba}
   Property P_PistonSurfaceB: Id {0a1f2ad1-d0b0-4c2d-ab96-5ea58f2ad315}
   Get Get: Id {57435720-e3ad-4686-b619-f1484e54ee8f}
   Property P_Position: Id {ecd4dedd-0cb4-4147-ba0a-08c9d58cd630}
   Get Get: Id {b618bc28-4b43-4b76-93ac-fcf905b068dd}
   Property P_PositionAbs: Id {209e36f6-751f-4240-9cf5-b9fb16eebcc3}
   Get Get: Id {c03056e5-e9cc-4e15-ba7e-aefbdeb24221}
   Property P_PressureChA: Id {471cd3ff-e656-456d-b21e-3fda36d5fa8a}
   Get Get: Id {a6241634-cb35-43cf-b205-078f1f07d390}
   Property P_PressureChB: Id {03707cd5-7bee-429d-8306-f3b3ddc5765c}
   Get Get: Id {6d6380ef-f945-459d-b206-fb36e7cb3fc0}
   Property P_PressureOk: Id {6b913370-94a9-471c-812d-bd6855387ffa}
   Get Get: Id {681e8f43-a680-471f-b3c8-f3cecc9ece1c}
   Property P_ReadyState: Id {1fa808d5-8df8-4027-bce1-4448834f347f}
   Get Get: Id {95333c44-72e4-4a9c-8f36-758f6a6c5354}
   Property P_SpeedInMmPerSecond: Id {7a045a39-f8cc-480e-bd59-c1f15e86d5cf}
   Get Get: Id {5cadc9e3-17f8-4fa6-95c8-fb62f2fe3e10}
   Property P_SpeedInPercent: Id {3fb7dbfa-2b1e-4209-a356-c8ba8ec22d25}
   Get Get: Id {c65ef769-845a-4360-a7b0-4e0c6016f632}
   Property P_StrokeLength: Id {8393f4e5-9e08-40fd-bea9-bcf7de5fb770}
   Get Get: Id {938b3200-55ce-46a1-89c0-542c0425c3cd}
   Property P_StrokeLengthInitialized: Id {9f06b182-b20c-4376-bcc5-f6911e48a611}
   Get Get: Id {02c02f9f-889f-4171-b3d9-7044a1afb128}
   Set Set: Id {14c6ee10-021d-49fd-a004-a11016f6c37d}
   Property P_WorkPressure: Id {076c9341-f880-4950-b6b0-64ccc401116c}
   Get Get: Id {e5ef4199-a585-48b5-ab0e-7eba9ef15b66} *)
